// TwinCAT 3 PLC project SDSPLC
// Title: SDS M2
// Company: Aperture Science
// Author: A. Wallace
// ProjectVersion: 0.0.0
// ProgramVersion: 3.1.4022.2
// libraries:
//   Tc2_Standard, * (Beckhoff Automation GmbH)
//   Tc2_System, * (Beckhoff Automation GmbH)
//   Tc3_Module, * (Beckhoff Automation GmbH)
//   LCLS General,0.1.2,SLAC
//   LCLSVacuumLib,1.12.6969,SLAC
//   Tc2_EtherCAT,3.3.13.0,Beckhoff Automation GmbH
//   Tc2_IoFunctions,3.3.11.0,Beckhoff Automation GmbH
//   Tc2_MC2,3.3.37.0,Beckhoff Automation GmbH
//   Tc2_ModbusSrv,3.3.1.0,Beckhoff Automation GmbH
//   Tc2_SerialCom,3.3.6.0,Beckhoff Automation GmbH
//   Tc2_SUPS,3.3.6.0,Beckhoff Automation GmbH
//   Tc2_Utilities,3.3.35.0,Beckhoff Automation GmbH
// project tree:
//   DUTs/ALI/ E_AxisMoveMode.TcDUT (not stored), E_CTRL_MODE.TcDUT (not stored), E_PropValveFBState.TcDUT (not stored), HMI_PropValveCtrlState.TcDUT (not stored), ST_ALI.TcDUT (not stored), ST_ManipAxis.TcDUT (not stored), ST_PIDParams.TcDUT (not stored), ST_PressureController.TcDUT (not stored), ST_PropValveMKS253.TcDUT (not stored)
//   DUTs/Bronkhorst/ E_BHElFlowUnit.TcDUT (not stored), ST_BhElFlow.TcDUT (not stored), ST_BhFMControl.TcDUT (not stored), ST_BhFMStatus.TcDUT (not stored)
//   DUTs/ E_AxisMotionState.TcDUT (not stored), ST_M3GasManifold.TcDUT (not stored), ST_ManifoldValve.TcDUT (not stored), ST_Proportionair.TcDUT (not stored), ST_RegDeadbandControls.TcDUT (not stored), ST_Regulator.TcDUT (not stored), ST_Selector.TcDUT (not stored), ST_SelectorM3.TcDUT (not stored), ST_SensirionFM.TcDUT (not stored), ST_Shaker.TcDUT (not stored), ST_ShakerControls.TcDUT (not stored)
//   DUTs/IO_Structs/ ST_ALIIO.TcDUT (not stored), ST_M2SelectorIO.TcDUT (not stored), ST_M3DeviceBaseIO.TcDUT (not stored), ST_M3GasManifoldIO.TcDUT (not stored), ST_M3PressCtrlIO.TcDUT (not stored), ST_M3SelectorIO.TcDUT (not stored)
//   DUTs/Sensirion/ ST_SensirionFMControl.TcDUT (not stored), ST_SensirionFMStatus.TcDUT (not stored)
//   DUTs/TEC/ ST_TECControl.TcDUT (not stored), ST_TECStatus.TcDUT (not stored)
//   DUTs/Vici/ ST_ViciControl.TcDUT (not stored), ST_ViciStatus.TcDUT (not stored)
//   GVLs/ GVL.TcGVL (not stored), GVL_Autosave.TcGVL (not stored), GVL_ComBuffers.TcGVL (not stored), GVL_Devices.TcGVL (not stored), GVL_IO.TcGVL (not stored), GVL_misc.TcGVL (not stored)
//   / PlcTask.TcTTO (not stored), SerialComm.TcTTO (not stored)
//   POUs/ALI/ FB_ALI.TcPOU (not stored), FB_PID_EXT.TcPOU (not stored), MC_SmoothMover.TcPOU (not stored), F_AxisRef_To_MSTA.TcPOU (not stored), FB_ManipAxis.TcPOU (not stored), FB_PropValve.TcPOU (not stored)
//   POUs/Bronkhorst/ FB_L01Driver.TcPOU (not stored), FB_FlowBusTransaction.TcPOU (not stored)
//   POUs/ FB_SelectorM3.TcPOU (not stored), MAIN.TcPOU (not stored), p_ALI.TcPOU (not stored), p_Autosave.TcPOU (not stored), p_AutoWash.TcPOU (not stored), p_CoolerShaker.TcPOU (not stored), p_ESTOP.TcPOU (not stored), p_Manifold.TcPOU (not stored), p_ModbusRx.TcPOU (not stored), p_ModbusTx.TcPOU (not stored), p_Regulators.TcPOU (not stored), p_SampleSelector.TcPOU (not stored), p_SampleSelector2.TcPOU (not stored), p_Shakers.TcPOU (not stored), p_SoftIO.TcPOU (not stored), p_VacGaugeSup.TcPOU (not stored), SerialTxRx.TcPOU (not stored), p_StatusLights.TcPOU (not stored)
//   POUs/Helpers/ FB_EcatDiag.TcPOU (not stored), FB_ManiValve.TcPOU (not stored), FB_SelectorSync.TcPOU (not stored), FB_ShiftByteArray.TcPOU (not stored)
//   POUs/Regulators/ FB_ProportionairRegulator.TcPOU (not stored), FB_Regulator.TcPOU (not stored), F_rPressure.TcPOU (not stored)
//   POUs/Sensirion/ FB_SensirionDriver.TcPOU (not stored), FB_SensirionTransaction.TcPOU (not stored), fSHDLCChecksum.TcPOU (not stored)
//   POUs/TEC/ FB_TECDriver.TcPOU (not stored), FB_TECTransaction.TcPOU (not stored)
//   POUs/VICI/ FB_ViciDriver.TcPOU, FB_ViciTransaction.TcPOU (not stored)
//   VISUs/ Main.TcVIS (not stored)
// real-time tasks:
//   TASK SerialComm: cycle T#5ms, priority 1, ADS port 350
//   TASK PlcTask: cycle T#10ms, priority 20, ADS port 351
// motion (NC):
// I/O:
//   DEVICE MAIN (EtherCAT)
// variable links:
//   SDSPLC Instance <-> MAIN (EtherCAT)
//     PlcTask Inputs/GVL.g_aEcatMaster1 <-> InfoData/AmsNetId
//     PlcTask Inputs/GVL_IO.iq_stPressCtrlA.i_SyncUnitWC <-> SyncUnits/[PCM A (EP1111)]/<unreferenced>/WcState/WcState
//   SDSPLC Instance <-> MAIN (EtherCAT)/ALI_Gauges (EP3174-0002)
//     PlcTask Inputs/GVL_Devices.stALI.i_EP3174_Ch{1..4} <-> AI Standard Channel {1..4}/Value  (4 links)
//   SDSPLC Instance <-> MAIN (EtherCAT)/ALI_PropValve (EP7041-0002)
//     PlcTask Inputs/GVL_Devices.stALI.stPropVlv.i_HLS <-> STM Status/Status/Digital input 1
//     PlcTask Inputs/GVL_Devices.stALI.stPropVlv.i_LLS <-> STM Status/Status/Digital input 2
//   SDSPLC Instance <-> MAIN (EtherCAT)/ALI_X (EP7041-0002)
//     PlcTask Inputs/GVL_Devices.stALI.axisX.xHiLS <-> STM Status/Status/Digital input 2
//     PlcTask Inputs/GVL_Devices.stALI.axisX.xLoLS <-> STM Status/Status/Digital input 1
//   SDSPLC Instance <-> MAIN (EtherCAT)/ALI_Y (EP7041-0002)
//     PlcTask Inputs/GVL_Devices.stALI.axisY.xHiLS <-> STM Status/Status/Digital input 2
//     PlcTask Inputs/GVL_Devices.stALI.axisY.xLoLS <-> STM Status/Status/Digital input 1
//   SDSPLC Instance <-> MAIN (EtherCAT)/ALI_Z (EP7041-0002)
//     PlcTask Inputs/GVL_Devices.stALI.axisZ.xHiLS <-> STM Status/Status/Digital input 2
//     PlcTask Inputs/GVL_Devices.stALI.axisZ.xLoLS <-> STM Status/Status/Digital input 1
//   SDSPLC Instance <-> MAIN (EtherCAT)/Gas_Mani_NeedleValve (EP4374-0002)
//     PlcTask Inputs/GVL_IO.iq_stM3GasManifold.i_EP4374_Ch1 <-> AI Inputs Channel 1/Value
//     PlcTask Inputs/GVL_IO.iq_stM3GasManifold.i_EP4374_Ch2 <-> AI Inputs Channel 2/Value
//     PlcTask Outputs/GVL_IO.iq_stM3GasManifold.q_EP4374_Ch3 <-> AO Outputs Channel 3/Analog output
//     PlcTask Outputs/GVL_IO.iq_stM3GasManifold.q_EP4374_Ch4 <-> AO Outputs Channel 4/Analog output
//   SDSPLC Instance <-> MAIN (EtherCAT)/Gas_Mani_ValveCtrl (EP2338-0001)
//     PlcTask Outputs/GVL_IO.iq_stM3GasManifold.q_EP2338_Ch{1..8} <-> Channel {9..16}/Output  (8 links)
//   SDSPLC Instance <-> MAIN (EtherCAT)/Gas_Mani_ValveRbk (EP2338-0001)
//     PlcTask Inputs/GVL_IO.iq_stM3GasManifold.i_EP2338_Ch{1..8} <-> Channel {1..8}/Input  (8 links)
//   SDSPLC Instance <-> MAIN (EtherCAT)/M2 Selector A (EP2338-0001)
//     PlcTask Inputs/GVL_IO.iq_stM2SelectorA.i_EP2338_Ch{5..8} <-> Channel {5..8}/Input  (4 links)
//     PlcTask Outputs/GVL_IO.iq_stM2SelectorA.q_EP2338_Ch{1..4} <-> Channel {9..12}/Output  (4 links)
//   SDSPLC Instance <-> MAIN (EtherCAT)/M2 Selector A (EP6002-0002)
//     SerialComm Inputs/GVL_IO.iq_stM2SelectorA.stComIn_EP6002P1/D[0] <-> COM TxPDO-Map Inputs Channel 1/Data In 0
//     SerialComm Inputs/GVL_IO.iq_stM2SelectorA.stComIn_EP6002P1/D[10] <-> COM TxPDO-Map Inputs Channel 1/Data In 10
//     SerialComm Inputs/GVL_IO.iq_stM2SelectorA.stComIn_EP6002P1/D[11] <-> COM TxPDO-Map Inputs Channel 1/Data In 11
//     SerialComm Inputs/GVL_IO.iq_stM2SelectorA.stComIn_EP6002P1/D[12] <-> COM TxPDO-Map Inputs Channel 1/Data In 12
//     SerialComm Inputs/GVL_IO.iq_stM2SelectorA.stComIn_EP6002P1/D[13] <-> COM TxPDO-Map Inputs Channel 1/Data In 13
//     SerialComm Inputs/GVL_IO.iq_stM2SelectorA.stComIn_EP6002P1/D[14] <-> COM TxPDO-Map Inputs Channel 1/Data In 14
//     SerialComm Inputs/GVL_IO.iq_stM2SelectorA.stComIn_EP6002P1/D[15] <-> COM TxPDO-Map Inputs Channel 1/Data In 15
//     SerialComm Inputs/GVL_IO.iq_stM2SelectorA.stComIn_EP6002P1/D[16] <-> COM TxPDO-Map Inputs Channel 1/Data In 16
//     SerialComm Inputs/GVL_IO.iq_stM2SelectorA.stComIn_EP6002P1/D[17] <-> COM TxPDO-Map Inputs Channel 1/Data In 17
//     SerialComm Inputs/GVL_IO.iq_stM2SelectorA.stComIn_EP6002P1/D[18] <-> COM TxPDO-Map Inputs Channel 1/Data In 18
//     SerialComm Inputs/GVL_IO.iq_stM2SelectorA.stComIn_EP6002P1/D[19] <-> COM TxPDO-Map Inputs Channel 1/Data In 19
//     SerialComm Inputs/GVL_IO.iq_stM2SelectorA.stComIn_EP6002P1/D[1] <-> COM TxPDO-Map Inputs Channel 1/Data In 1
//     SerialComm Inputs/GVL_IO.iq_stM2SelectorA.stComIn_EP6002P1/D[20] <-> COM TxPDO-Map Inputs Channel 1/Data In 20
//     SerialComm Inputs/GVL_IO.iq_stM2SelectorA.stComIn_EP6002P1/D[21] <-> COM TxPDO-Map Inputs Channel 1/Data In 21
//     SerialComm Inputs/GVL_IO.iq_stM2SelectorA.stComIn_EP6002P1/D[2] <-> COM TxPDO-Map Inputs Channel 1/Data In 2
//     SerialComm Inputs/GVL_IO.iq_stM2SelectorA.stComIn_EP6002P1/D[3] <-> COM TxPDO-Map Inputs Channel 1/Data In 3
//     SerialComm Inputs/GVL_IO.iq_stM2SelectorA.stComIn_EP6002P1/D[4] <-> COM TxPDO-Map Inputs Channel 1/Data In 4
//     SerialComm Inputs/GVL_IO.iq_stM2SelectorA.stComIn_EP6002P1/D[5] <-> COM TxPDO-Map Inputs Channel 1/Data In 5
//     SerialComm Inputs/GVL_IO.iq_stM2SelectorA.stComIn_EP6002P1/D[6] <-> COM TxPDO-Map Inputs Channel 1/Data In 6
//     SerialComm Inputs/GVL_IO.iq_stM2SelectorA.stComIn_EP6002P1/D[7] <-> COM TxPDO-Map Inputs Channel 1/Data In 7
//     SerialComm Inputs/GVL_IO.iq_stM2SelectorA.stComIn_EP6002P1/D[8] <-> COM TxPDO-Map Inputs Channel 1/Data In 8
//     SerialComm Inputs/GVL_IO.iq_stM2SelectorA.stComIn_EP6002P1/D[9] <-> COM TxPDO-Map Inputs Channel 1/Data In 9
//     SerialComm Inputs/GVL_IO.iq_stM2SelectorA.stComIn_EP6002P2/D[0] <-> COM TxPDO-Map Inputs Channel 2/Data In 0
//     SerialComm Inputs/GVL_IO.iq_stM2SelectorA.stComIn_EP6002P2/D[10] <-> COM TxPDO-Map Inputs Channel 2/Data In 10
//     SerialComm Inputs/GVL_IO.iq_stM2SelectorA.stComIn_EP6002P2/D[11] <-> COM TxPDO-Map Inputs Channel 2/Data In 11
//     SerialComm Inputs/GVL_IO.iq_stM2SelectorA.stComIn_EP6002P2/D[12] <-> COM TxPDO-Map Inputs Channel 2/Data In 12
//     SerialComm Inputs/GVL_IO.iq_stM2SelectorA.stComIn_EP6002P2/D[13] <-> COM TxPDO-Map Inputs Channel 2/Data In 13
//     SerialComm Inputs/GVL_IO.iq_stM2SelectorA.stComIn_EP6002P2/D[14] <-> COM TxPDO-Map Inputs Channel 2/Data In 14
//     SerialComm Inputs/GVL_IO.iq_stM2SelectorA.stComIn_EP6002P2/D[15] <-> COM TxPDO-Map Inputs Channel 2/Data In 15
//     SerialComm Inputs/GVL_IO.iq_stM2SelectorA.stComIn_EP6002P2/D[16] <-> COM TxPDO-Map Inputs Channel 2/Data In 16
//     SerialComm Inputs/GVL_IO.iq_stM2SelectorA.stComIn_EP6002P2/D[17] <-> COM TxPDO-Map Inputs Channel 2/Data In 17
//     SerialComm Inputs/GVL_IO.iq_stM2SelectorA.stComIn_EP6002P2/D[18] <-> COM TxPDO-Map Inputs Channel 2/Data In 18
//     SerialComm Inputs/GVL_IO.iq_stM2SelectorA.stComIn_EP6002P2/D[19] <-> COM TxPDO-Map Inputs Channel 2/Data In 19
//     SerialComm Inputs/GVL_IO.iq_stM2SelectorA.stComIn_EP6002P2/D[1] <-> COM TxPDO-Map Inputs Channel 2/Data In 1
//     SerialComm Inputs/GVL_IO.iq_stM2SelectorA.stComIn_EP6002P2/D[20] <-> COM TxPDO-Map Inputs Channel 2/Data In 20
//     SerialComm Inputs/GVL_IO.iq_stM2SelectorA.stComIn_EP6002P2/D[21] <-> COM TxPDO-Map Inputs Channel 2/Data In 21
//     SerialComm Inputs/GVL_IO.iq_stM2SelectorA.stComIn_EP6002P2/D[2] <-> COM TxPDO-Map Inputs Channel 2/Data In 2
//     SerialComm Inputs/GVL_IO.iq_stM2SelectorA.stComIn_EP6002P2/D[3] <-> COM TxPDO-Map Inputs Channel 2/Data In 3
//     SerialComm Inputs/GVL_IO.iq_stM2SelectorA.stComIn_EP6002P2/D[4] <-> COM TxPDO-Map Inputs Channel 2/Data In 4
//     SerialComm Inputs/GVL_IO.iq_stM2SelectorA.stComIn_EP6002P2/D[5] <-> COM TxPDO-Map Inputs Channel 2/Data In 5
//     SerialComm Inputs/GVL_IO.iq_stM2SelectorA.stComIn_EP6002P2/D[6] <-> COM TxPDO-Map Inputs Channel 2/Data In 6
//     SerialComm Inputs/GVL_IO.iq_stM2SelectorA.stComIn_EP6002P2/D[7] <-> COM TxPDO-Map Inputs Channel 2/Data In 7
//     SerialComm Inputs/GVL_IO.iq_stM2SelectorA.stComIn_EP6002P2/D[8] <-> COM TxPDO-Map Inputs Channel 2/Data In 8
//     SerialComm Inputs/GVL_IO.iq_stM2SelectorA.stComIn_EP6002P2/D[9] <-> COM TxPDO-Map Inputs Channel 2/Data In 9
//     SerialComm Inputs/GVL_IO.iq_stM2SelectorA.stComIn_EP6002P1/Status <-> COM TxPDO-Map Inputs Channel 1/Status
//     SerialComm Inputs/GVL_IO.iq_stM2SelectorA.stComIn_EP6002P2/Status <-> COM TxPDO-Map Inputs Channel 2/Status
//     SerialComm Outputs/GVL_IO.iq_stM2SelectorA.stComOut_EP6002P1/Ctrl <-> COM RxPDO-Map Outputs Channel 1/Ctrl
//     SerialComm Outputs/GVL_IO.iq_stM2SelectorA.stComOut_EP6002P2/Ctrl <-> COM RxPDO-Map Outputs Channel 2/Ctrl
//     SerialComm Outputs/GVL_IO.iq_stM2SelectorA.stComOut_EP6002P1/D[0] <-> COM RxPDO-Map Outputs Channel 1/Data Out 0
//     SerialComm Outputs/GVL_IO.iq_stM2SelectorA.stComOut_EP6002P1/D[10] <-> COM RxPDO-Map Outputs Channel 1/Data Out 10
//     SerialComm Outputs/GVL_IO.iq_stM2SelectorA.stComOut_EP6002P1/D[11] <-> COM RxPDO-Map Outputs Channel 1/Data Out 11
//     SerialComm Outputs/GVL_IO.iq_stM2SelectorA.stComOut_EP6002P1/D[12] <-> COM RxPDO-Map Outputs Channel 1/Data Out 12
//     SerialComm Outputs/GVL_IO.iq_stM2SelectorA.stComOut_EP6002P1/D[13] <-> COM RxPDO-Map Outputs Channel 1/Data Out 13
//     SerialComm Outputs/GVL_IO.iq_stM2SelectorA.stComOut_EP6002P1/D[14] <-> COM RxPDO-Map Outputs Channel 1/Data Out 14
//     SerialComm Outputs/GVL_IO.iq_stM2SelectorA.stComOut_EP6002P1/D[15] <-> COM RxPDO-Map Outputs Channel 1/Data Out 15
//     SerialComm Outputs/GVL_IO.iq_stM2SelectorA.stComOut_EP6002P1/D[16] <-> COM RxPDO-Map Outputs Channel 1/Data Out 16
//     SerialComm Outputs/GVL_IO.iq_stM2SelectorA.stComOut_EP6002P1/D[17] <-> COM RxPDO-Map Outputs Channel 1/Data Out 17
//     SerialComm Outputs/GVL_IO.iq_stM2SelectorA.stComOut_EP6002P1/D[18] <-> COM RxPDO-Map Outputs Channel 1/Data Out 18
//     SerialComm Outputs/GVL_IO.iq_stM2SelectorA.stComOut_EP6002P1/D[19] <-> COM RxPDO-Map Outputs Channel 1/Data Out 19
//     SerialComm Outputs/GVL_IO.iq_stM2SelectorA.stComOut_EP6002P1/D[1] <-> COM RxPDO-Map Outputs Channel 1/Data Out 1
//     SerialComm Outputs/GVL_IO.iq_stM2SelectorA.stComOut_EP6002P1/D[20] <-> COM RxPDO-Map Outputs Channel 1/Data Out 20
//     SerialComm Outputs/GVL_IO.iq_stM2SelectorA.stComOut_EP6002P1/D[21] <-> COM RxPDO-Map Outputs Channel 1/Data Out 21
//     SerialComm Outputs/GVL_IO.iq_stM2SelectorA.stComOut_EP6002P1/D[2] <-> COM RxPDO-Map Outputs Channel 1/Data Out 2
//     SerialComm Outputs/GVL_IO.iq_stM2SelectorA.stComOut_EP6002P1/D[3] <-> COM RxPDO-Map Outputs Channel 1/Data Out 3
//     SerialComm Outputs/GVL_IO.iq_stM2SelectorA.stComOut_EP6002P1/D[4] <-> COM RxPDO-Map Outputs Channel 1/Data Out 4
//     SerialComm Outputs/GVL_IO.iq_stM2SelectorA.stComOut_EP6002P1/D[5] <-> COM RxPDO-Map Outputs Channel 1/Data Out 5
//     SerialComm Outputs/GVL_IO.iq_stM2SelectorA.stComOut_EP6002P1/D[6] <-> COM RxPDO-Map Outputs Channel 1/Data Out 6
//     SerialComm Outputs/GVL_IO.iq_stM2SelectorA.stComOut_EP6002P1/D[7] <-> COM RxPDO-Map Outputs Channel 1/Data Out 7
//     SerialComm Outputs/GVL_IO.iq_stM2SelectorA.stComOut_EP6002P1/D[8] <-> COM RxPDO-Map Outputs Channel 1/Data Out 8
//     SerialComm Outputs/GVL_IO.iq_stM2SelectorA.stComOut_EP6002P1/D[9] <-> COM RxPDO-Map Outputs Channel 1/Data Out 9
//     SerialComm Outputs/GVL_IO.iq_stM2SelectorA.stComOut_EP6002P2/D[0] <-> COM RxPDO-Map Outputs Channel 2/Data Out 0
//     SerialComm Outputs/GVL_IO.iq_stM2SelectorA.stComOut_EP6002P2/D[10] <-> COM RxPDO-Map Outputs Channel 2/Data Out 10
//     SerialComm Outputs/GVL_IO.iq_stM2SelectorA.stComOut_EP6002P2/D[11] <-> COM RxPDO-Map Outputs Channel 2/Data Out 11
//     SerialComm Outputs/GVL_IO.iq_stM2SelectorA.stComOut_EP6002P2/D[12] <-> COM RxPDO-Map Outputs Channel 2/Data Out 12
//     SerialComm Outputs/GVL_IO.iq_stM2SelectorA.stComOut_EP6002P2/D[13] <-> COM RxPDO-Map Outputs Channel 2/Data Out 13
//     SerialComm Outputs/GVL_IO.iq_stM2SelectorA.stComOut_EP6002P2/D[14] <-> COM RxPDO-Map Outputs Channel 2/Data Out 14
//     SerialComm Outputs/GVL_IO.iq_stM2SelectorA.stComOut_EP6002P2/D[15] <-> COM RxPDO-Map Outputs Channel 2/Data Out 15
//     SerialComm Outputs/GVL_IO.iq_stM2SelectorA.stComOut_EP6002P2/D[16] <-> COM RxPDO-Map Outputs Channel 2/Data Out 16
//     SerialComm Outputs/GVL_IO.iq_stM2SelectorA.stComOut_EP6002P2/D[17] <-> COM RxPDO-Map Outputs Channel 2/Data Out 17
//     SerialComm Outputs/GVL_IO.iq_stM2SelectorA.stComOut_EP6002P2/D[18] <-> COM RxPDO-Map Outputs Channel 2/Data Out 18
//     SerialComm Outputs/GVL_IO.iq_stM2SelectorA.stComOut_EP6002P2/D[19] <-> COM RxPDO-Map Outputs Channel 2/Data Out 19
//     SerialComm Outputs/GVL_IO.iq_stM2SelectorA.stComOut_EP6002P2/D[1] <-> COM RxPDO-Map Outputs Channel 2/Data Out 1
//     SerialComm Outputs/GVL_IO.iq_stM2SelectorA.stComOut_EP6002P2/D[20] <-> COM RxPDO-Map Outputs Channel 2/Data Out 20
//     SerialComm Outputs/GVL_IO.iq_stM2SelectorA.stComOut_EP6002P2/D[21] <-> COM RxPDO-Map Outputs Channel 2/Data Out 21
//     SerialComm Outputs/GVL_IO.iq_stM2SelectorA.stComOut_EP6002P2/D[2] <-> COM RxPDO-Map Outputs Channel 2/Data Out 2
//     SerialComm Outputs/GVL_IO.iq_stM2SelectorA.stComOut_EP6002P2/D[3] <-> COM RxPDO-Map Outputs Channel 2/Data Out 3
//     SerialComm Outputs/GVL_IO.iq_stM2SelectorA.stComOut_EP6002P2/D[4] <-> COM RxPDO-Map Outputs Channel 2/Data Out 4
//     SerialComm Outputs/GVL_IO.iq_stM2SelectorA.stComOut_EP6002P2/D[5] <-> COM RxPDO-Map Outputs Channel 2/Data Out 5
//     SerialComm Outputs/GVL_IO.iq_stM2SelectorA.stComOut_EP6002P2/D[6] <-> COM RxPDO-Map Outputs Channel 2/Data Out 6
//     SerialComm Outputs/GVL_IO.iq_stM2SelectorA.stComOut_EP6002P2/D[7] <-> COM RxPDO-Map Outputs Channel 2/Data Out 7
//     SerialComm Outputs/GVL_IO.iq_stM2SelectorA.stComOut_EP6002P2/D[8] <-> COM RxPDO-Map Outputs Channel 2/Data Out 8
//     SerialComm Outputs/GVL_IO.iq_stM2SelectorA.stComOut_EP6002P2/D[9] <-> COM RxPDO-Map Outputs Channel 2/Data Out 9
//   SDSPLC Instance <-> MAIN (EtherCAT)/M2 Selector B (EP2338-0001)
//     PlcTask Inputs/GVL_IO.iq_stM2SelectorB.i_EP2338_Ch{5..8} <-> Channel {5..8}/Input  (4 links)
//     PlcTask Outputs/GVL_IO.iq_stM2SelectorB.q_EP2338_Ch{1..4} <-> Channel {9..12}/Output  (4 links)
//   SDSPLC Instance <-> MAIN (EtherCAT)/M2 Selector B (EP6002-0002)
//     SerialComm Inputs/GVL_IO.iq_stM2SelectorB.stComIn_EP6002P1/D[0] <-> COM TxPDO-Map Inputs Channel 1/Data In 0
//     SerialComm Inputs/GVL_IO.iq_stM2SelectorB.stComIn_EP6002P1/D[10] <-> COM TxPDO-Map Inputs Channel 1/Data In 10
//     SerialComm Inputs/GVL_IO.iq_stM2SelectorB.stComIn_EP6002P1/D[11] <-> COM TxPDO-Map Inputs Channel 1/Data In 11
//     SerialComm Inputs/GVL_IO.iq_stM2SelectorB.stComIn_EP6002P1/D[12] <-> COM TxPDO-Map Inputs Channel 1/Data In 12
//     SerialComm Inputs/GVL_IO.iq_stM2SelectorB.stComIn_EP6002P1/D[13] <-> COM TxPDO-Map Inputs Channel 1/Data In 13
//     SerialComm Inputs/GVL_IO.iq_stM2SelectorB.stComIn_EP6002P1/D[14] <-> COM TxPDO-Map Inputs Channel 1/Data In 14
//     SerialComm Inputs/GVL_IO.iq_stM2SelectorB.stComIn_EP6002P1/D[15] <-> COM TxPDO-Map Inputs Channel 1/Data In 15
//     SerialComm Inputs/GVL_IO.iq_stM2SelectorB.stComIn_EP6002P1/D[16] <-> COM TxPDO-Map Inputs Channel 1/Data In 16
//     SerialComm Inputs/GVL_IO.iq_stM2SelectorB.stComIn_EP6002P1/D[17] <-> COM TxPDO-Map Inputs Channel 1/Data In 17
//     SerialComm Inputs/GVL_IO.iq_stM2SelectorB.stComIn_EP6002P1/D[18] <-> COM TxPDO-Map Inputs Channel 1/Data In 18
//     SerialComm Inputs/GVL_IO.iq_stM2SelectorB.stComIn_EP6002P1/D[19] <-> COM TxPDO-Map Inputs Channel 1/Data In 19
//     SerialComm Inputs/GVL_IO.iq_stM2SelectorB.stComIn_EP6002P1/D[1] <-> COM TxPDO-Map Inputs Channel 1/Data In 1
//     SerialComm Inputs/GVL_IO.iq_stM2SelectorB.stComIn_EP6002P1/D[20] <-> COM TxPDO-Map Inputs Channel 1/Data In 20
//     SerialComm Inputs/GVL_IO.iq_stM2SelectorB.stComIn_EP6002P1/D[21] <-> COM TxPDO-Map Inputs Channel 1/Data In 21
//     SerialComm Inputs/GVL_IO.iq_stM2SelectorB.stComIn_EP6002P1/D[2] <-> COM TxPDO-Map Inputs Channel 1/Data In 2
//     SerialComm Inputs/GVL_IO.iq_stM2SelectorB.stComIn_EP6002P1/D[3] <-> COM TxPDO-Map Inputs Channel 1/Data In 3
//     SerialComm Inputs/GVL_IO.iq_stM2SelectorB.stComIn_EP6002P1/D[4] <-> COM TxPDO-Map Inputs Channel 1/Data In 4
//     SerialComm Inputs/GVL_IO.iq_stM2SelectorB.stComIn_EP6002P1/D[5] <-> COM TxPDO-Map Inputs Channel 1/Data In 5
//     SerialComm Inputs/GVL_IO.iq_stM2SelectorB.stComIn_EP6002P1/D[6] <-> COM TxPDO-Map Inputs Channel 1/Data In 6
//     SerialComm Inputs/GVL_IO.iq_stM2SelectorB.stComIn_EP6002P1/D[7] <-> COM TxPDO-Map Inputs Channel 1/Data In 7
//     SerialComm Inputs/GVL_IO.iq_stM2SelectorB.stComIn_EP6002P1/D[8] <-> COM TxPDO-Map Inputs Channel 1/Data In 8
//     SerialComm Inputs/GVL_IO.iq_stM2SelectorB.stComIn_EP6002P1/D[9] <-> COM TxPDO-Map Inputs Channel 1/Data In 9
//     SerialComm Inputs/GVL_IO.iq_stM2SelectorB.stComIn_EP6002P2/D[0] <-> COM TxPDO-Map Inputs Channel 2/Data In 0
//     SerialComm Inputs/GVL_IO.iq_stM2SelectorB.stComIn_EP6002P2/D[10] <-> COM TxPDO-Map Inputs Channel 2/Data In 10
//     SerialComm Inputs/GVL_IO.iq_stM2SelectorB.stComIn_EP6002P2/D[11] <-> COM TxPDO-Map Inputs Channel 2/Data In 11
//     SerialComm Inputs/GVL_IO.iq_stM2SelectorB.stComIn_EP6002P2/D[12] <-> COM TxPDO-Map Inputs Channel 2/Data In 12
//     SerialComm Inputs/GVL_IO.iq_stM2SelectorB.stComIn_EP6002P2/D[13] <-> COM TxPDO-Map Inputs Channel 2/Data In 13
//     SerialComm Inputs/GVL_IO.iq_stM2SelectorB.stComIn_EP6002P2/D[14] <-> COM TxPDO-Map Inputs Channel 2/Data In 14
//     SerialComm Inputs/GVL_IO.iq_stM2SelectorB.stComIn_EP6002P2/D[15] <-> COM TxPDO-Map Inputs Channel 2/Data In 15
//     SerialComm Inputs/GVL_IO.iq_stM2SelectorB.stComIn_EP6002P2/D[16] <-> COM TxPDO-Map Inputs Channel 2/Data In 16
//     SerialComm Inputs/GVL_IO.iq_stM2SelectorB.stComIn_EP6002P2/D[17] <-> COM TxPDO-Map Inputs Channel 2/Data In 17
//     SerialComm Inputs/GVL_IO.iq_stM2SelectorB.stComIn_EP6002P2/D[18] <-> COM TxPDO-Map Inputs Channel 2/Data In 18
//     SerialComm Inputs/GVL_IO.iq_stM2SelectorB.stComIn_EP6002P2/D[19] <-> COM TxPDO-Map Inputs Channel 2/Data In 19
//     SerialComm Inputs/GVL_IO.iq_stM2SelectorB.stComIn_EP6002P2/D[1] <-> COM TxPDO-Map Inputs Channel 2/Data In 1
//     SerialComm Inputs/GVL_IO.iq_stM2SelectorB.stComIn_EP6002P2/D[20] <-> COM TxPDO-Map Inputs Channel 2/Data In 20
//     SerialComm Inputs/GVL_IO.iq_stM2SelectorB.stComIn_EP6002P2/D[21] <-> COM TxPDO-Map Inputs Channel 2/Data In 21
//     SerialComm Inputs/GVL_IO.iq_stM2SelectorB.stComIn_EP6002P2/D[2] <-> COM TxPDO-Map Inputs Channel 2/Data In 2
//     SerialComm Inputs/GVL_IO.iq_stM2SelectorB.stComIn_EP6002P2/D[3] <-> COM TxPDO-Map Inputs Channel 2/Data In 3
//     SerialComm Inputs/GVL_IO.iq_stM2SelectorB.stComIn_EP6002P2/D[4] <-> COM TxPDO-Map Inputs Channel 2/Data In 4
//     SerialComm Inputs/GVL_IO.iq_stM2SelectorB.stComIn_EP6002P2/D[5] <-> COM TxPDO-Map Inputs Channel 2/Data In 5
//     SerialComm Inputs/GVL_IO.iq_stM2SelectorB.stComIn_EP6002P2/D[6] <-> COM TxPDO-Map Inputs Channel 2/Data In 6
//     SerialComm Inputs/GVL_IO.iq_stM2SelectorB.stComIn_EP6002P2/D[7] <-> COM TxPDO-Map Inputs Channel 2/Data In 7
//     SerialComm Inputs/GVL_IO.iq_stM2SelectorB.stComIn_EP6002P2/D[8] <-> COM TxPDO-Map Inputs Channel 2/Data In 8
//     SerialComm Inputs/GVL_IO.iq_stM2SelectorB.stComIn_EP6002P2/D[9] <-> COM TxPDO-Map Inputs Channel 2/Data In 9
//     SerialComm Inputs/GVL_IO.iq_stM2SelectorB.stComIn_EP6002P1/Status <-> COM TxPDO-Map Inputs Channel 1/Status
//     SerialComm Inputs/GVL_IO.iq_stM2SelectorB.stComIn_EP6002P2/Status <-> COM TxPDO-Map Inputs Channel 2/Status
//     SerialComm Outputs/GVL_IO.iq_stM2SelectorB.stComOut_EP6002P1/Ctrl <-> COM RxPDO-Map Outputs Channel 1/Ctrl
//     SerialComm Outputs/GVL_IO.iq_stM2SelectorB.stComOut_EP6002P2/Ctrl <-> COM RxPDO-Map Outputs Channel 2/Ctrl
//     SerialComm Outputs/GVL_IO.iq_stM2SelectorB.stComOut_EP6002P1/D[0] <-> COM RxPDO-Map Outputs Channel 1/Data Out 0
//     SerialComm Outputs/GVL_IO.iq_stM2SelectorB.stComOut_EP6002P1/D[10] <-> COM RxPDO-Map Outputs Channel 1/Data Out 10
//     SerialComm Outputs/GVL_IO.iq_stM2SelectorB.stComOut_EP6002P1/D[11] <-> COM RxPDO-Map Outputs Channel 1/Data Out 11
//     SerialComm Outputs/GVL_IO.iq_stM2SelectorB.stComOut_EP6002P1/D[12] <-> COM RxPDO-Map Outputs Channel 1/Data Out 12
//     SerialComm Outputs/GVL_IO.iq_stM2SelectorB.stComOut_EP6002P1/D[13] <-> COM RxPDO-Map Outputs Channel 1/Data Out 13
//     SerialComm Outputs/GVL_IO.iq_stM2SelectorB.stComOut_EP6002P1/D[14] <-> COM RxPDO-Map Outputs Channel 1/Data Out 14
//     SerialComm Outputs/GVL_IO.iq_stM2SelectorB.stComOut_EP6002P1/D[15] <-> COM RxPDO-Map Outputs Channel 1/Data Out 15
//     SerialComm Outputs/GVL_IO.iq_stM2SelectorB.stComOut_EP6002P1/D[16] <-> COM RxPDO-Map Outputs Channel 1/Data Out 16
//     SerialComm Outputs/GVL_IO.iq_stM2SelectorB.stComOut_EP6002P1/D[17] <-> COM RxPDO-Map Outputs Channel 1/Data Out 17
//     SerialComm Outputs/GVL_IO.iq_stM2SelectorB.stComOut_EP6002P1/D[18] <-> COM RxPDO-Map Outputs Channel 1/Data Out 18
//     SerialComm Outputs/GVL_IO.iq_stM2SelectorB.stComOut_EP6002P1/D[19] <-> COM RxPDO-Map Outputs Channel 1/Data Out 19
//     SerialComm Outputs/GVL_IO.iq_stM2SelectorB.stComOut_EP6002P1/D[1] <-> COM RxPDO-Map Outputs Channel 1/Data Out 1
//     SerialComm Outputs/GVL_IO.iq_stM2SelectorB.stComOut_EP6002P1/D[20] <-> COM RxPDO-Map Outputs Channel 1/Data Out 20
//     SerialComm Outputs/GVL_IO.iq_stM2SelectorB.stComOut_EP6002P1/D[21] <-> COM RxPDO-Map Outputs Channel 1/Data Out 21
//     SerialComm Outputs/GVL_IO.iq_stM2SelectorB.stComOut_EP6002P1/D[2] <-> COM RxPDO-Map Outputs Channel 1/Data Out 2
//     SerialComm Outputs/GVL_IO.iq_stM2SelectorB.stComOut_EP6002P1/D[3] <-> COM RxPDO-Map Outputs Channel 1/Data Out 3
//     SerialComm Outputs/GVL_IO.iq_stM2SelectorB.stComOut_EP6002P1/D[4] <-> COM RxPDO-Map Outputs Channel 1/Data Out 4
//     SerialComm Outputs/GVL_IO.iq_stM2SelectorB.stComOut_EP6002P1/D[5] <-> COM RxPDO-Map Outputs Channel 1/Data Out 5
//     SerialComm Outputs/GVL_IO.iq_stM2SelectorB.stComOut_EP6002P1/D[6] <-> COM RxPDO-Map Outputs Channel 1/Data Out 6
//     SerialComm Outputs/GVL_IO.iq_stM2SelectorB.stComOut_EP6002P1/D[7] <-> COM RxPDO-Map Outputs Channel 1/Data Out 7
//     SerialComm Outputs/GVL_IO.iq_stM2SelectorB.stComOut_EP6002P1/D[8] <-> COM RxPDO-Map Outputs Channel 1/Data Out 8
//     SerialComm Outputs/GVL_IO.iq_stM2SelectorB.stComOut_EP6002P1/D[9] <-> COM RxPDO-Map Outputs Channel 1/Data Out 9
//     SerialComm Outputs/GVL_IO.iq_stM2SelectorB.stComOut_EP6002P2/D[0] <-> COM RxPDO-Map Outputs Channel 2/Data Out 0
//     SerialComm Outputs/GVL_IO.iq_stM2SelectorB.stComOut_EP6002P2/D[10] <-> COM RxPDO-Map Outputs Channel 2/Data Out 10
//     SerialComm Outputs/GVL_IO.iq_stM2SelectorB.stComOut_EP6002P2/D[11] <-> COM RxPDO-Map Outputs Channel 2/Data Out 11
//     SerialComm Outputs/GVL_IO.iq_stM2SelectorB.stComOut_EP6002P2/D[12] <-> COM RxPDO-Map Outputs Channel 2/Data Out 12
//     SerialComm Outputs/GVL_IO.iq_stM2SelectorB.stComOut_EP6002P2/D[13] <-> COM RxPDO-Map Outputs Channel 2/Data Out 13
//     SerialComm Outputs/GVL_IO.iq_stM2SelectorB.stComOut_EP6002P2/D[14] <-> COM RxPDO-Map Outputs Channel 2/Data Out 14
//     SerialComm Outputs/GVL_IO.iq_stM2SelectorB.stComOut_EP6002P2/D[15] <-> COM RxPDO-Map Outputs Channel 2/Data Out 15
//     SerialComm Outputs/GVL_IO.iq_stM2SelectorB.stComOut_EP6002P2/D[16] <-> COM RxPDO-Map Outputs Channel 2/Data Out 16
//     SerialComm Outputs/GVL_IO.iq_stM2SelectorB.stComOut_EP6002P2/D[17] <-> COM RxPDO-Map Outputs Channel 2/Data Out 17
//     SerialComm Outputs/GVL_IO.iq_stM2SelectorB.stComOut_EP6002P2/D[18] <-> COM RxPDO-Map Outputs Channel 2/Data Out 18
//     SerialComm Outputs/GVL_IO.iq_stM2SelectorB.stComOut_EP6002P2/D[19] <-> COM RxPDO-Map Outputs Channel 2/Data Out 19
//     SerialComm Outputs/GVL_IO.iq_stM2SelectorB.stComOut_EP6002P2/D[1] <-> COM RxPDO-Map Outputs Channel 2/Data Out 1
//     SerialComm Outputs/GVL_IO.iq_stM2SelectorB.stComOut_EP6002P2/D[20] <-> COM RxPDO-Map Outputs Channel 2/Data Out 20
//     SerialComm Outputs/GVL_IO.iq_stM2SelectorB.stComOut_EP6002P2/D[21] <-> COM RxPDO-Map Outputs Channel 2/Data Out 21
//     SerialComm Outputs/GVL_IO.iq_stM2SelectorB.stComOut_EP6002P2/D[2] <-> COM RxPDO-Map Outputs Channel 2/Data Out 2
//     SerialComm Outputs/GVL_IO.iq_stM2SelectorB.stComOut_EP6002P2/D[3] <-> COM RxPDO-Map Outputs Channel 2/Data Out 3
//     SerialComm Outputs/GVL_IO.iq_stM2SelectorB.stComOut_EP6002P2/D[4] <-> COM RxPDO-Map Outputs Channel 2/Data Out 4
//     SerialComm Outputs/GVL_IO.iq_stM2SelectorB.stComOut_EP6002P2/D[5] <-> COM RxPDO-Map Outputs Channel 2/Data Out 5
//     SerialComm Outputs/GVL_IO.iq_stM2SelectorB.stComOut_EP6002P2/D[6] <-> COM RxPDO-Map Outputs Channel 2/Data Out 6
//     SerialComm Outputs/GVL_IO.iq_stM2SelectorB.stComOut_EP6002P2/D[7] <-> COM RxPDO-Map Outputs Channel 2/Data Out 7
//     SerialComm Outputs/GVL_IO.iq_stM2SelectorB.stComOut_EP6002P2/D[8] <-> COM RxPDO-Map Outputs Channel 2/Data Out 8
//     SerialComm Outputs/GVL_IO.iq_stM2SelectorB.stComOut_EP6002P2/D[9] <-> COM RxPDO-Map Outputs Channel 2/Data Out 9
//   SDSPLC Instance <-> MAIN (EtherCAT)/M3 Selector A Digital IO (EP2338-1001)
//     PlcTask Inputs/GVL_IO.iq_stM3SelectorA.i_EP2338_Ch{5..8} <-> Channel {5..8}/Input  (4 links)
//     PlcTask Outputs/GVL_IO.iq_stM3SelectorA.q_EP2338_Ch{1..4} <-> Channel {9..12}/Output  (4 links)
//   SDSPLC Instance <-> MAIN (EtherCAT)/M3 Selector A Mass Flow Meter (Mass Flow / Pressure Controller - Slave)
//     PlcTask Inputs/GVL_IO.iq_stM3SelectorA.i_RawUnit <-> TxPDO/Unit
//     PlcTask Inputs/GVL_IO.iq_stM3SelectorA.i_mfmFlow <-> TxPDO/fMeasure
//   SDSPLC Instance <-> MAIN (EtherCAT)/M3 Selector A Serial IO (EP6002-0002)
//     PlcTask Inputs/GVL_IO.iq_stM3SelectorA.stComIn_EP6002P1/D[0] <-> COM TxPDO-Map Inputs Channel 1/Data In 0
//     PlcTask Inputs/GVL_IO.iq_stM3SelectorA.stComIn_EP6002P1/D[10] <-> COM TxPDO-Map Inputs Channel 1/Data In 10
//     PlcTask Inputs/GVL_IO.iq_stM3SelectorA.stComIn_EP6002P1/D[11] <-> COM TxPDO-Map Inputs Channel 1/Data In 11
//     PlcTask Inputs/GVL_IO.iq_stM3SelectorA.stComIn_EP6002P1/D[12] <-> COM TxPDO-Map Inputs Channel 1/Data In 12
//     PlcTask Inputs/GVL_IO.iq_stM3SelectorA.stComIn_EP6002P1/D[13] <-> COM TxPDO-Map Inputs Channel 1/Data In 13
//     PlcTask Inputs/GVL_IO.iq_stM3SelectorA.stComIn_EP6002P1/D[14] <-> COM TxPDO-Map Inputs Channel 1/Data In 14
//     PlcTask Inputs/GVL_IO.iq_stM3SelectorA.stComIn_EP6002P1/D[15] <-> COM TxPDO-Map Inputs Channel 1/Data In 15
//     PlcTask Inputs/GVL_IO.iq_stM3SelectorA.stComIn_EP6002P1/D[16] <-> COM TxPDO-Map Inputs Channel 1/Data In 16
//     PlcTask Inputs/GVL_IO.iq_stM3SelectorA.stComIn_EP6002P1/D[17] <-> COM TxPDO-Map Inputs Channel 1/Data In 17
//     PlcTask Inputs/GVL_IO.iq_stM3SelectorA.stComIn_EP6002P1/D[18] <-> COM TxPDO-Map Inputs Channel 1/Data In 18
//     PlcTask Inputs/GVL_IO.iq_stM3SelectorA.stComIn_EP6002P1/D[19] <-> COM TxPDO-Map Inputs Channel 1/Data In 19
//     PlcTask Inputs/GVL_IO.iq_stM3SelectorA.stComIn_EP6002P1/D[1] <-> COM TxPDO-Map Inputs Channel 1/Data In 1
//     PlcTask Inputs/GVL_IO.iq_stM3SelectorA.stComIn_EP6002P1/D[20] <-> COM TxPDO-Map Inputs Channel 1/Data In 20
//     PlcTask Inputs/GVL_IO.iq_stM3SelectorA.stComIn_EP6002P1/D[21] <-> COM TxPDO-Map Inputs Channel 1/Data In 21
//     PlcTask Inputs/GVL_IO.iq_stM3SelectorA.stComIn_EP6002P1/D[2] <-> COM TxPDO-Map Inputs Channel 1/Data In 2
//     PlcTask Inputs/GVL_IO.iq_stM3SelectorA.stComIn_EP6002P1/D[3] <-> COM TxPDO-Map Inputs Channel 1/Data In 3
//     PlcTask Inputs/GVL_IO.iq_stM3SelectorA.stComIn_EP6002P1/D[4] <-> COM TxPDO-Map Inputs Channel 1/Data In 4
//     PlcTask Inputs/GVL_IO.iq_stM3SelectorA.stComIn_EP6002P1/D[5] <-> COM TxPDO-Map Inputs Channel 1/Data In 5
//     PlcTask Inputs/GVL_IO.iq_stM3SelectorA.stComIn_EP6002P1/D[6] <-> COM TxPDO-Map Inputs Channel 1/Data In 6
//     PlcTask Inputs/GVL_IO.iq_stM3SelectorA.stComIn_EP6002P1/D[7] <-> COM TxPDO-Map Inputs Channel 1/Data In 7
//     PlcTask Inputs/GVL_IO.iq_stM3SelectorA.stComIn_EP6002P1/D[8] <-> COM TxPDO-Map Inputs Channel 1/Data In 8
//     PlcTask Inputs/GVL_IO.iq_stM3SelectorA.stComIn_EP6002P1/D[9] <-> COM TxPDO-Map Inputs Channel 1/Data In 9
//     PlcTask Inputs/GVL_IO.iq_stM3SelectorA.stComIn_EP6002P2/D[0] <-> COM TxPDO-Map Inputs Channel 2/Data In 0
//     PlcTask Inputs/GVL_IO.iq_stM3SelectorA.stComIn_EP6002P2/D[10] <-> COM TxPDO-Map Inputs Channel 2/Data In 10
//     PlcTask Inputs/GVL_IO.iq_stM3SelectorA.stComIn_EP6002P2/D[11] <-> COM TxPDO-Map Inputs Channel 2/Data In 11
//     PlcTask Inputs/GVL_IO.iq_stM3SelectorA.stComIn_EP6002P2/D[12] <-> COM TxPDO-Map Inputs Channel 2/Data In 12
//     PlcTask Inputs/GVL_IO.iq_stM3SelectorA.stComIn_EP6002P2/D[13] <-> COM TxPDO-Map Inputs Channel 2/Data In 13
//     PlcTask Inputs/GVL_IO.iq_stM3SelectorA.stComIn_EP6002P2/D[14] <-> COM TxPDO-Map Inputs Channel 2/Data In 14
//     PlcTask Inputs/GVL_IO.iq_stM3SelectorA.stComIn_EP6002P2/D[15] <-> COM TxPDO-Map Inputs Channel 2/Data In 15
//     PlcTask Inputs/GVL_IO.iq_stM3SelectorA.stComIn_EP6002P2/D[16] <-> COM TxPDO-Map Inputs Channel 2/Data In 16
//     PlcTask Inputs/GVL_IO.iq_stM3SelectorA.stComIn_EP6002P2/D[17] <-> COM TxPDO-Map Inputs Channel 2/Data In 17
//     PlcTask Inputs/GVL_IO.iq_stM3SelectorA.stComIn_EP6002P2/D[18] <-> COM TxPDO-Map Inputs Channel 2/Data In 18
//     PlcTask Inputs/GVL_IO.iq_stM3SelectorA.stComIn_EP6002P2/D[19] <-> COM TxPDO-Map Inputs Channel 2/Data In 19
//     PlcTask Inputs/GVL_IO.iq_stM3SelectorA.stComIn_EP6002P2/D[1] <-> COM TxPDO-Map Inputs Channel 2/Data In 1
//     PlcTask Inputs/GVL_IO.iq_stM3SelectorA.stComIn_EP6002P2/D[20] <-> COM TxPDO-Map Inputs Channel 2/Data In 20
//     PlcTask Inputs/GVL_IO.iq_stM3SelectorA.stComIn_EP6002P2/D[21] <-> COM TxPDO-Map Inputs Channel 2/Data In 21
//     PlcTask Inputs/GVL_IO.iq_stM3SelectorA.stComIn_EP6002P2/D[2] <-> COM TxPDO-Map Inputs Channel 2/Data In 2
//     PlcTask Inputs/GVL_IO.iq_stM3SelectorA.stComIn_EP6002P2/D[3] <-> COM TxPDO-Map Inputs Channel 2/Data In 3
//     PlcTask Inputs/GVL_IO.iq_stM3SelectorA.stComIn_EP6002P2/D[4] <-> COM TxPDO-Map Inputs Channel 2/Data In 4
//     PlcTask Inputs/GVL_IO.iq_stM3SelectorA.stComIn_EP6002P2/D[5] <-> COM TxPDO-Map Inputs Channel 2/Data In 5
//     PlcTask Inputs/GVL_IO.iq_stM3SelectorA.stComIn_EP6002P2/D[6] <-> COM TxPDO-Map Inputs Channel 2/Data In 6
//     PlcTask Inputs/GVL_IO.iq_stM3SelectorA.stComIn_EP6002P2/D[7] <-> COM TxPDO-Map Inputs Channel 2/Data In 7
//     PlcTask Inputs/GVL_IO.iq_stM3SelectorA.stComIn_EP6002P2/D[8] <-> COM TxPDO-Map Inputs Channel 2/Data In 8
//     PlcTask Inputs/GVL_IO.iq_stM3SelectorA.stComIn_EP6002P2/D[9] <-> COM TxPDO-Map Inputs Channel 2/Data In 9
//     PlcTask Inputs/GVL_IO.iq_stM3SelectorA.stComIn_EP6002P1/Status <-> COM TxPDO-Map Inputs Channel 1/Status
//     PlcTask Inputs/GVL_IO.iq_stM3SelectorA.stComIn_EP6002P2/Status <-> COM TxPDO-Map Inputs Channel 2/Status
//     PlcTask Outputs/GVL_IO.iq_stM3SelectorA.stComOut_EP6002P1/Ctrl <-> COM RxPDO-Map Outputs Channel 1/Ctrl
//     PlcTask Outputs/GVL_IO.iq_stM3SelectorA.stComOut_EP6002P2/Ctrl <-> COM RxPDO-Map Outputs Channel 2/Ctrl
//     PlcTask Outputs/GVL_IO.iq_stM3SelectorA.stComOut_EP6002P1/D[0] <-> COM RxPDO-Map Outputs Channel 1/Data Out 0
//     PlcTask Outputs/GVL_IO.iq_stM3SelectorA.stComOut_EP6002P1/D[10] <-> COM RxPDO-Map Outputs Channel 1/Data Out 10
//     PlcTask Outputs/GVL_IO.iq_stM3SelectorA.stComOut_EP6002P1/D[11] <-> COM RxPDO-Map Outputs Channel 1/Data Out 11
//     PlcTask Outputs/GVL_IO.iq_stM3SelectorA.stComOut_EP6002P1/D[12] <-> COM RxPDO-Map Outputs Channel 1/Data Out 12
//     PlcTask Outputs/GVL_IO.iq_stM3SelectorA.stComOut_EP6002P1/D[13] <-> COM RxPDO-Map Outputs Channel 1/Data Out 13
//     PlcTask Outputs/GVL_IO.iq_stM3SelectorA.stComOut_EP6002P1/D[14] <-> COM RxPDO-Map Outputs Channel 1/Data Out 14
//     PlcTask Outputs/GVL_IO.iq_stM3SelectorA.stComOut_EP6002P1/D[15] <-> COM RxPDO-Map Outputs Channel 1/Data Out 15
//     PlcTask Outputs/GVL_IO.iq_stM3SelectorA.stComOut_EP6002P1/D[16] <-> COM RxPDO-Map Outputs Channel 1/Data Out 16
//     PlcTask Outputs/GVL_IO.iq_stM3SelectorA.stComOut_EP6002P1/D[17] <-> COM RxPDO-Map Outputs Channel 1/Data Out 17
//     PlcTask Outputs/GVL_IO.iq_stM3SelectorA.stComOut_EP6002P1/D[18] <-> COM RxPDO-Map Outputs Channel 1/Data Out 18
//     PlcTask Outputs/GVL_IO.iq_stM3SelectorA.stComOut_EP6002P1/D[19] <-> COM RxPDO-Map Outputs Channel 1/Data Out 19
//     PlcTask Outputs/GVL_IO.iq_stM3SelectorA.stComOut_EP6002P1/D[1] <-> COM RxPDO-Map Outputs Channel 1/Data Out 1
//     PlcTask Outputs/GVL_IO.iq_stM3SelectorA.stComOut_EP6002P1/D[20] <-> COM RxPDO-Map Outputs Channel 1/Data Out 20
//     PlcTask Outputs/GVL_IO.iq_stM3SelectorA.stComOut_EP6002P1/D[21] <-> COM RxPDO-Map Outputs Channel 1/Data Out 21
//     PlcTask Outputs/GVL_IO.iq_stM3SelectorA.stComOut_EP6002P1/D[2] <-> COM RxPDO-Map Outputs Channel 1/Data Out 2
//     PlcTask Outputs/GVL_IO.iq_stM3SelectorA.stComOut_EP6002P1/D[3] <-> COM RxPDO-Map Outputs Channel 1/Data Out 3
//     PlcTask Outputs/GVL_IO.iq_stM3SelectorA.stComOut_EP6002P1/D[4] <-> COM RxPDO-Map Outputs Channel 1/Data Out 4
//     PlcTask Outputs/GVL_IO.iq_stM3SelectorA.stComOut_EP6002P1/D[5] <-> COM RxPDO-Map Outputs Channel 1/Data Out 5
//     PlcTask Outputs/GVL_IO.iq_stM3SelectorA.stComOut_EP6002P1/D[6] <-> COM RxPDO-Map Outputs Channel 1/Data Out 6
//     PlcTask Outputs/GVL_IO.iq_stM3SelectorA.stComOut_EP6002P1/D[7] <-> COM RxPDO-Map Outputs Channel 1/Data Out 7
//     PlcTask Outputs/GVL_IO.iq_stM3SelectorA.stComOut_EP6002P1/D[8] <-> COM RxPDO-Map Outputs Channel 1/Data Out 8
//     PlcTask Outputs/GVL_IO.iq_stM3SelectorA.stComOut_EP6002P1/D[9] <-> COM RxPDO-Map Outputs Channel 1/Data Out 9
//     PlcTask Outputs/GVL_IO.iq_stM3SelectorA.stComOut_EP6002P2/D[0] <-> COM RxPDO-Map Outputs Channel 2/Data Out 0
//     PlcTask Outputs/GVL_IO.iq_stM3SelectorA.stComOut_EP6002P2/D[10] <-> COM RxPDO-Map Outputs Channel 2/Data Out 10
//     PlcTask Outputs/GVL_IO.iq_stM3SelectorA.stComOut_EP6002P2/D[11] <-> COM RxPDO-Map Outputs Channel 2/Data Out 11
//     PlcTask Outputs/GVL_IO.iq_stM3SelectorA.stComOut_EP6002P2/D[12] <-> COM RxPDO-Map Outputs Channel 2/Data Out 12
//     PlcTask Outputs/GVL_IO.iq_stM3SelectorA.stComOut_EP6002P2/D[13] <-> COM RxPDO-Map Outputs Channel 2/Data Out 13
//     PlcTask Outputs/GVL_IO.iq_stM3SelectorA.stComOut_EP6002P2/D[14] <-> COM RxPDO-Map Outputs Channel 2/Data Out 14
//     PlcTask Outputs/GVL_IO.iq_stM3SelectorA.stComOut_EP6002P2/D[15] <-> COM RxPDO-Map Outputs Channel 2/Data Out 15
//     PlcTask Outputs/GVL_IO.iq_stM3SelectorA.stComOut_EP6002P2/D[16] <-> COM RxPDO-Map Outputs Channel 2/Data Out 16
//     PlcTask Outputs/GVL_IO.iq_stM3SelectorA.stComOut_EP6002P2/D[17] <-> COM RxPDO-Map Outputs Channel 2/Data Out 17
//     PlcTask Outputs/GVL_IO.iq_stM3SelectorA.stComOut_EP6002P2/D[18] <-> COM RxPDO-Map Outputs Channel 2/Data Out 18
//     PlcTask Outputs/GVL_IO.iq_stM3SelectorA.stComOut_EP6002P2/D[19] <-> COM RxPDO-Map Outputs Channel 2/Data Out 19
//     PlcTask Outputs/GVL_IO.iq_stM3SelectorA.stComOut_EP6002P2/D[1] <-> COM RxPDO-Map Outputs Channel 2/Data Out 1
//     PlcTask Outputs/GVL_IO.iq_stM3SelectorA.stComOut_EP6002P2/D[20] <-> COM RxPDO-Map Outputs Channel 2/Data Out 20
//     PlcTask Outputs/GVL_IO.iq_stM3SelectorA.stComOut_EP6002P2/D[21] <-> COM RxPDO-Map Outputs Channel 2/Data Out 21
//     PlcTask Outputs/GVL_IO.iq_stM3SelectorA.stComOut_EP6002P2/D[2] <-> COM RxPDO-Map Outputs Channel 2/Data Out 2
//     PlcTask Outputs/GVL_IO.iq_stM3SelectorA.stComOut_EP6002P2/D[3] <-> COM RxPDO-Map Outputs Channel 2/Data Out 3
//     PlcTask Outputs/GVL_IO.iq_stM3SelectorA.stComOut_EP6002P2/D[4] <-> COM RxPDO-Map Outputs Channel 2/Data Out 4
//     PlcTask Outputs/GVL_IO.iq_stM3SelectorA.stComOut_EP6002P2/D[5] <-> COM RxPDO-Map Outputs Channel 2/Data Out 5
//     PlcTask Outputs/GVL_IO.iq_stM3SelectorA.stComOut_EP6002P2/D[6] <-> COM RxPDO-Map Outputs Channel 2/Data Out 6
//     PlcTask Outputs/GVL_IO.iq_stM3SelectorA.stComOut_EP6002P2/D[7] <-> COM RxPDO-Map Outputs Channel 2/Data Out 7
//     PlcTask Outputs/GVL_IO.iq_stM3SelectorA.stComOut_EP6002P2/D[8] <-> COM RxPDO-Map Outputs Channel 2/Data Out 8
//     PlcTask Outputs/GVL_IO.iq_stM3SelectorA.stComOut_EP6002P2/D[9] <-> COM RxPDO-Map Outputs Channel 2/Data Out 9
//   SDSPLC Instance <-> MAIN (EtherCAT)/M3 Selector B Digital IO (EP2338-1001)
//     PlcTask Inputs/GVL_IO.iq_stM3SelectorB.i_EP2338_Ch{5..8} <-> Channel {5..8}/Input  (4 links)
//     PlcTask Outputs/GVL_IO.iq_stM3SelectorB.q_EP2338_Ch{1..4} <-> Channel {9..12}/Output  (4 links)
//   SDSPLC Instance <-> MAIN (EtherCAT)/M3 Selector B Mass Flow Meter (Mass Flow / Pressure Controller - Slave)
//     PlcTask Inputs/GVL_IO.iq_stM3SelectorB.i_RawUnit <-> TxPDO/Unit
//     PlcTask Inputs/GVL_IO.iq_stM3SelectorB.i_mfmFlow <-> TxPDO/fMeasure
//   SDSPLC Instance <-> MAIN (EtherCAT)/M3 Selector B Serial IO (EP6002-0002)
//     PlcTask Inputs/GVL_IO.iq_stM3SelectorB.stComIn_EP6002P1/D[0] <-> COM TxPDO-Map Inputs Channel 1/Data In 0
//     PlcTask Inputs/GVL_IO.iq_stM3SelectorB.stComIn_EP6002P1/D[10] <-> COM TxPDO-Map Inputs Channel 1/Data In 10
//     PlcTask Inputs/GVL_IO.iq_stM3SelectorB.stComIn_EP6002P1/D[11] <-> COM TxPDO-Map Inputs Channel 1/Data In 11
//     PlcTask Inputs/GVL_IO.iq_stM3SelectorB.stComIn_EP6002P1/D[12] <-> COM TxPDO-Map Inputs Channel 1/Data In 12
//     PlcTask Inputs/GVL_IO.iq_stM3SelectorB.stComIn_EP6002P1/D[13] <-> COM TxPDO-Map Inputs Channel 1/Data In 13
//     PlcTask Inputs/GVL_IO.iq_stM3SelectorB.stComIn_EP6002P1/D[14] <-> COM TxPDO-Map Inputs Channel 1/Data In 14
//     PlcTask Inputs/GVL_IO.iq_stM3SelectorB.stComIn_EP6002P1/D[15] <-> COM TxPDO-Map Inputs Channel 1/Data In 15
//     PlcTask Inputs/GVL_IO.iq_stM3SelectorB.stComIn_EP6002P1/D[16] <-> COM TxPDO-Map Inputs Channel 1/Data In 16
//     PlcTask Inputs/GVL_IO.iq_stM3SelectorB.stComIn_EP6002P1/D[17] <-> COM TxPDO-Map Inputs Channel 1/Data In 17
//     PlcTask Inputs/GVL_IO.iq_stM3SelectorB.stComIn_EP6002P1/D[18] <-> COM TxPDO-Map Inputs Channel 1/Data In 18
//     PlcTask Inputs/GVL_IO.iq_stM3SelectorB.stComIn_EP6002P1/D[19] <-> COM TxPDO-Map Inputs Channel 1/Data In 19
//     PlcTask Inputs/GVL_IO.iq_stM3SelectorB.stComIn_EP6002P1/D[1] <-> COM TxPDO-Map Inputs Channel 1/Data In 1
//     PlcTask Inputs/GVL_IO.iq_stM3SelectorB.stComIn_EP6002P1/D[20] <-> COM TxPDO-Map Inputs Channel 1/Data In 20
//     PlcTask Inputs/GVL_IO.iq_stM3SelectorB.stComIn_EP6002P1/D[21] <-> COM TxPDO-Map Inputs Channel 1/Data In 21
//     PlcTask Inputs/GVL_IO.iq_stM3SelectorB.stComIn_EP6002P1/D[2] <-> COM TxPDO-Map Inputs Channel 1/Data In 2
//     PlcTask Inputs/GVL_IO.iq_stM3SelectorB.stComIn_EP6002P1/D[3] <-> COM TxPDO-Map Inputs Channel 1/Data In 3
//     PlcTask Inputs/GVL_IO.iq_stM3SelectorB.stComIn_EP6002P1/D[4] <-> COM TxPDO-Map Inputs Channel 1/Data In 4
//     PlcTask Inputs/GVL_IO.iq_stM3SelectorB.stComIn_EP6002P1/D[5] <-> COM TxPDO-Map Inputs Channel 1/Data In 5
//     PlcTask Inputs/GVL_IO.iq_stM3SelectorB.stComIn_EP6002P1/D[6] <-> COM TxPDO-Map Inputs Channel 1/Data In 6
//     PlcTask Inputs/GVL_IO.iq_stM3SelectorB.stComIn_EP6002P1/D[7] <-> COM TxPDO-Map Inputs Channel 1/Data In 7
//     PlcTask Inputs/GVL_IO.iq_stM3SelectorB.stComIn_EP6002P1/D[8] <-> COM TxPDO-Map Inputs Channel 1/Data In 8
//     PlcTask Inputs/GVL_IO.iq_stM3SelectorB.stComIn_EP6002P1/D[9] <-> COM TxPDO-Map Inputs Channel 1/Data In 9
//     PlcTask Inputs/GVL_IO.iq_stM3SelectorB.stComIn_EP6002P2/D[0] <-> COM TxPDO-Map Inputs Channel 2/Data In 0
//     PlcTask Inputs/GVL_IO.iq_stM3SelectorB.stComIn_EP6002P2/D[10] <-> COM TxPDO-Map Inputs Channel 2/Data In 10
//     PlcTask Inputs/GVL_IO.iq_stM3SelectorB.stComIn_EP6002P2/D[11] <-> COM TxPDO-Map Inputs Channel 2/Data In 11
//     PlcTask Inputs/GVL_IO.iq_stM3SelectorB.stComIn_EP6002P2/D[12] <-> COM TxPDO-Map Inputs Channel 2/Data In 12
//     PlcTask Inputs/GVL_IO.iq_stM3SelectorB.stComIn_EP6002P2/D[13] <-> COM TxPDO-Map Inputs Channel 2/Data In 13
//     PlcTask Inputs/GVL_IO.iq_stM3SelectorB.stComIn_EP6002P2/D[14] <-> COM TxPDO-Map Inputs Channel 2/Data In 14
//     PlcTask Inputs/GVL_IO.iq_stM3SelectorB.stComIn_EP6002P2/D[15] <-> COM TxPDO-Map Inputs Channel 2/Data In 15
//     PlcTask Inputs/GVL_IO.iq_stM3SelectorB.stComIn_EP6002P2/D[16] <-> COM TxPDO-Map Inputs Channel 2/Data In 16
//     PlcTask Inputs/GVL_IO.iq_stM3SelectorB.stComIn_EP6002P2/D[17] <-> COM TxPDO-Map Inputs Channel 2/Data In 17
//     PlcTask Inputs/GVL_IO.iq_stM3SelectorB.stComIn_EP6002P2/D[18] <-> COM TxPDO-Map Inputs Channel 2/Data In 18
//     PlcTask Inputs/GVL_IO.iq_stM3SelectorB.stComIn_EP6002P2/D[19] <-> COM TxPDO-Map Inputs Channel 2/Data In 19
//     PlcTask Inputs/GVL_IO.iq_stM3SelectorB.stComIn_EP6002P2/D[1] <-> COM TxPDO-Map Inputs Channel 2/Data In 1
//     PlcTask Inputs/GVL_IO.iq_stM3SelectorB.stComIn_EP6002P2/D[20] <-> COM TxPDO-Map Inputs Channel 2/Data In 20
//     PlcTask Inputs/GVL_IO.iq_stM3SelectorB.stComIn_EP6002P2/D[21] <-> COM TxPDO-Map Inputs Channel 2/Data In 21
//     PlcTask Inputs/GVL_IO.iq_stM3SelectorB.stComIn_EP6002P2/D[2] <-> COM TxPDO-Map Inputs Channel 2/Data In 2
//     PlcTask Inputs/GVL_IO.iq_stM3SelectorB.stComIn_EP6002P2/D[3] <-> COM TxPDO-Map Inputs Channel 2/Data In 3
//     PlcTask Inputs/GVL_IO.iq_stM3SelectorB.stComIn_EP6002P2/D[4] <-> COM TxPDO-Map Inputs Channel 2/Data In 4
//     PlcTask Inputs/GVL_IO.iq_stM3SelectorB.stComIn_EP6002P2/D[5] <-> COM TxPDO-Map Inputs Channel 2/Data In 5
//     PlcTask Inputs/GVL_IO.iq_stM3SelectorB.stComIn_EP6002P2/D[6] <-> COM TxPDO-Map Inputs Channel 2/Data In 6
//     PlcTask Inputs/GVL_IO.iq_stM3SelectorB.stComIn_EP6002P2/D[7] <-> COM TxPDO-Map Inputs Channel 2/Data In 7
//     PlcTask Inputs/GVL_IO.iq_stM3SelectorB.stComIn_EP6002P2/D[8] <-> COM TxPDO-Map Inputs Channel 2/Data In 8
//     PlcTask Inputs/GVL_IO.iq_stM3SelectorB.stComIn_EP6002P2/D[9] <-> COM TxPDO-Map Inputs Channel 2/Data In 9
//     PlcTask Inputs/GVL_IO.iq_stM3SelectorB.stComIn_EP6002P1/Status <-> COM TxPDO-Map Inputs Channel 1/Status
//     PlcTask Inputs/GVL_IO.iq_stM3SelectorB.stComIn_EP6002P2/Status <-> COM TxPDO-Map Inputs Channel 2/Status
//     PlcTask Outputs/GVL_IO.iq_stM3SelectorB.stComOut_EP6002P1/Ctrl <-> COM RxPDO-Map Outputs Channel 1/Ctrl
//     PlcTask Outputs/GVL_IO.iq_stM3SelectorB.stComOut_EP6002P2/Ctrl <-> COM RxPDO-Map Outputs Channel 2/Ctrl
//     PlcTask Outputs/GVL_IO.iq_stM3SelectorB.stComOut_EP6002P1/D[0] <-> COM RxPDO-Map Outputs Channel 1/Data Out 0
//     PlcTask Outputs/GVL_IO.iq_stM3SelectorB.stComOut_EP6002P1/D[10] <-> COM RxPDO-Map Outputs Channel 1/Data Out 10
//     PlcTask Outputs/GVL_IO.iq_stM3SelectorB.stComOut_EP6002P1/D[11] <-> COM RxPDO-Map Outputs Channel 1/Data Out 11
//     PlcTask Outputs/GVL_IO.iq_stM3SelectorB.stComOut_EP6002P1/D[12] <-> COM RxPDO-Map Outputs Channel 1/Data Out 12
//     PlcTask Outputs/GVL_IO.iq_stM3SelectorB.stComOut_EP6002P1/D[13] <-> COM RxPDO-Map Outputs Channel 1/Data Out 13
//     PlcTask Outputs/GVL_IO.iq_stM3SelectorB.stComOut_EP6002P1/D[14] <-> COM RxPDO-Map Outputs Channel 1/Data Out 14
//     PlcTask Outputs/GVL_IO.iq_stM3SelectorB.stComOut_EP6002P1/D[15] <-> COM RxPDO-Map Outputs Channel 1/Data Out 15
//     PlcTask Outputs/GVL_IO.iq_stM3SelectorB.stComOut_EP6002P1/D[16] <-> COM RxPDO-Map Outputs Channel 1/Data Out 16
//     PlcTask Outputs/GVL_IO.iq_stM3SelectorB.stComOut_EP6002P1/D[17] <-> COM RxPDO-Map Outputs Channel 1/Data Out 17
//     PlcTask Outputs/GVL_IO.iq_stM3SelectorB.stComOut_EP6002P1/D[18] <-> COM RxPDO-Map Outputs Channel 1/Data Out 18
//     PlcTask Outputs/GVL_IO.iq_stM3SelectorB.stComOut_EP6002P1/D[19] <-> COM RxPDO-Map Outputs Channel 1/Data Out 19
//     PlcTask Outputs/GVL_IO.iq_stM3SelectorB.stComOut_EP6002P1/D[1] <-> COM RxPDO-Map Outputs Channel 1/Data Out 1
//     PlcTask Outputs/GVL_IO.iq_stM3SelectorB.stComOut_EP6002P1/D[20] <-> COM RxPDO-Map Outputs Channel 1/Data Out 20
//     PlcTask Outputs/GVL_IO.iq_stM3SelectorB.stComOut_EP6002P1/D[21] <-> COM RxPDO-Map Outputs Channel 1/Data Out 21
//     PlcTask Outputs/GVL_IO.iq_stM3SelectorB.stComOut_EP6002P1/D[2] <-> COM RxPDO-Map Outputs Channel 1/Data Out 2
//     PlcTask Outputs/GVL_IO.iq_stM3SelectorB.stComOut_EP6002P1/D[3] <-> COM RxPDO-Map Outputs Channel 1/Data Out 3
//     PlcTask Outputs/GVL_IO.iq_stM3SelectorB.stComOut_EP6002P1/D[4] <-> COM RxPDO-Map Outputs Channel 1/Data Out 4
//     PlcTask Outputs/GVL_IO.iq_stM3SelectorB.stComOut_EP6002P1/D[5] <-> COM RxPDO-Map Outputs Channel 1/Data Out 5
//     PlcTask Outputs/GVL_IO.iq_stM3SelectorB.stComOut_EP6002P1/D[6] <-> COM RxPDO-Map Outputs Channel 1/Data Out 6
//     PlcTask Outputs/GVL_IO.iq_stM3SelectorB.stComOut_EP6002P1/D[7] <-> COM RxPDO-Map Outputs Channel 1/Data Out 7
//     PlcTask Outputs/GVL_IO.iq_stM3SelectorB.stComOut_EP6002P1/D[8] <-> COM RxPDO-Map Outputs Channel 1/Data Out 8
//     PlcTask Outputs/GVL_IO.iq_stM3SelectorB.stComOut_EP6002P1/D[9] <-> COM RxPDO-Map Outputs Channel 1/Data Out 9
//     PlcTask Outputs/GVL_IO.iq_stM3SelectorB.stComOut_EP6002P2/D[0] <-> COM RxPDO-Map Outputs Channel 2/Data Out 0
//     PlcTask Outputs/GVL_IO.iq_stM3SelectorB.stComOut_EP6002P2/D[10] <-> COM RxPDO-Map Outputs Channel 2/Data Out 10
//     PlcTask Outputs/GVL_IO.iq_stM3SelectorB.stComOut_EP6002P2/D[11] <-> COM RxPDO-Map Outputs Channel 2/Data Out 11
//     PlcTask Outputs/GVL_IO.iq_stM3SelectorB.stComOut_EP6002P2/D[12] <-> COM RxPDO-Map Outputs Channel 2/Data Out 12
//     PlcTask Outputs/GVL_IO.iq_stM3SelectorB.stComOut_EP6002P2/D[13] <-> COM RxPDO-Map Outputs Channel 2/Data Out 13
//     PlcTask Outputs/GVL_IO.iq_stM3SelectorB.stComOut_EP6002P2/D[14] <-> COM RxPDO-Map Outputs Channel 2/Data Out 14
//     PlcTask Outputs/GVL_IO.iq_stM3SelectorB.stComOut_EP6002P2/D[15] <-> COM RxPDO-Map Outputs Channel 2/Data Out 15
//     PlcTask Outputs/GVL_IO.iq_stM3SelectorB.stComOut_EP6002P2/D[16] <-> COM RxPDO-Map Outputs Channel 2/Data Out 16
//     PlcTask Outputs/GVL_IO.iq_stM3SelectorB.stComOut_EP6002P2/D[17] <-> COM RxPDO-Map Outputs Channel 2/Data Out 17
//     PlcTask Outputs/GVL_IO.iq_stM3SelectorB.stComOut_EP6002P2/D[18] <-> COM RxPDO-Map Outputs Channel 2/Data Out 18
//     PlcTask Outputs/GVL_IO.iq_stM3SelectorB.stComOut_EP6002P2/D[19] <-> COM RxPDO-Map Outputs Channel 2/Data Out 19
//     PlcTask Outputs/GVL_IO.iq_stM3SelectorB.stComOut_EP6002P2/D[1] <-> COM RxPDO-Map Outputs Channel 2/Data Out 1
//     PlcTask Outputs/GVL_IO.iq_stM3SelectorB.stComOut_EP6002P2/D[20] <-> COM RxPDO-Map Outputs Channel 2/Data Out 20
//     PlcTask Outputs/GVL_IO.iq_stM3SelectorB.stComOut_EP6002P2/D[21] <-> COM RxPDO-Map Outputs Channel 2/Data Out 21
//     PlcTask Outputs/GVL_IO.iq_stM3SelectorB.stComOut_EP6002P2/D[2] <-> COM RxPDO-Map Outputs Channel 2/Data Out 2
//     PlcTask Outputs/GVL_IO.iq_stM3SelectorB.stComOut_EP6002P2/D[3] <-> COM RxPDO-Map Outputs Channel 2/Data Out 3
//     PlcTask Outputs/GVL_IO.iq_stM3SelectorB.stComOut_EP6002P2/D[4] <-> COM RxPDO-Map Outputs Channel 2/Data Out 4
//     PlcTask Outputs/GVL_IO.iq_stM3SelectorB.stComOut_EP6002P2/D[5] <-> COM RxPDO-Map Outputs Channel 2/Data Out 5
//     PlcTask Outputs/GVL_IO.iq_stM3SelectorB.stComOut_EP6002P2/D[6] <-> COM RxPDO-Map Outputs Channel 2/Data Out 6
//     PlcTask Outputs/GVL_IO.iq_stM3SelectorB.stComOut_EP6002P2/D[7] <-> COM RxPDO-Map Outputs Channel 2/Data Out 7
//     PlcTask Outputs/GVL_IO.iq_stM3SelectorB.stComOut_EP6002P2/D[8] <-> COM RxPDO-Map Outputs Channel 2/Data Out 8
//     PlcTask Outputs/GVL_IO.iq_stM3SelectorB.stComOut_EP6002P2/D[9] <-> COM RxPDO-Map Outputs Channel 2/Data Out 9
//   SDSPLC Instance <-> MAIN (EtherCAT)/PCM A (EP3174-0002)
//     PlcTask Inputs/GVL_IO.iq_stPressCtrlA.i_EP3174_Ch{1..4} <-> AI Standard Channel {1..4}/Value  (4 links)
//   SDSPLC Instance <-> MAIN (EtherCAT)/PCM A (EP4374-0002)
//     PlcTask Inputs/GVL_IO.iq_stPressCtrlA.i_EP4374_Ch1 <-> AI Inputs Channel 1/Value
//     PlcTask Inputs/GVL_IO.iq_stPressCtrlA.i_EP4374_Ch2 <-> AI Inputs Channel 2/Value
//     PlcTask Outputs/GVL_IO.iq_stPressCtrlA.q_EP4374_Ch3 <-> AO Outputs Channel 3/Analog output
//     PlcTask Outputs/GVL_IO.iq_stPressCtrlA.q_EP4374_Ch4 <-> AO Outputs Channel 4/Analog output
//   SDSPLC Instance <-> MAIN (EtherCAT)/PCM A (EP6002-0002)
//     PlcTask Inputs/GVL_IO.iq_stPressCtrlA.stComIn_EP6002P1/D[0] <-> COM TxPDO-Map Inputs Channel 1/Data In 0
//     PlcTask Inputs/GVL_IO.iq_stPressCtrlA.stComIn_EP6002P1/D[10] <-> COM TxPDO-Map Inputs Channel 1/Data In 10
//     PlcTask Inputs/GVL_IO.iq_stPressCtrlA.stComIn_EP6002P1/D[11] <-> COM TxPDO-Map Inputs Channel 1/Data In 11
//     PlcTask Inputs/GVL_IO.iq_stPressCtrlA.stComIn_EP6002P1/D[12] <-> COM TxPDO-Map Inputs Channel 1/Data In 12
//     PlcTask Inputs/GVL_IO.iq_stPressCtrlA.stComIn_EP6002P1/D[13] <-> COM TxPDO-Map Inputs Channel 1/Data In 13
//     PlcTask Inputs/GVL_IO.iq_stPressCtrlA.stComIn_EP6002P1/D[14] <-> COM TxPDO-Map Inputs Channel 1/Data In 14
//     PlcTask Inputs/GVL_IO.iq_stPressCtrlA.stComIn_EP6002P1/D[15] <-> COM TxPDO-Map Inputs Channel 1/Data In 15
//     PlcTask Inputs/GVL_IO.iq_stPressCtrlA.stComIn_EP6002P1/D[16] <-> COM TxPDO-Map Inputs Channel 1/Data In 16
//     PlcTask Inputs/GVL_IO.iq_stPressCtrlA.stComIn_EP6002P1/D[17] <-> COM TxPDO-Map Inputs Channel 1/Data In 17
//     PlcTask Inputs/GVL_IO.iq_stPressCtrlA.stComIn_EP6002P1/D[18] <-> COM TxPDO-Map Inputs Channel 1/Data In 18
//     PlcTask Inputs/GVL_IO.iq_stPressCtrlA.stComIn_EP6002P1/D[19] <-> COM TxPDO-Map Inputs Channel 1/Data In 19
//     PlcTask Inputs/GVL_IO.iq_stPressCtrlA.stComIn_EP6002P1/D[1] <-> COM TxPDO-Map Inputs Channel 1/Data In 1
//     PlcTask Inputs/GVL_IO.iq_stPressCtrlA.stComIn_EP6002P1/D[20] <-> COM TxPDO-Map Inputs Channel 1/Data In 20
//     PlcTask Inputs/GVL_IO.iq_stPressCtrlA.stComIn_EP6002P1/D[21] <-> COM TxPDO-Map Inputs Channel 1/Data In 21
//     PlcTask Inputs/GVL_IO.iq_stPressCtrlA.stComIn_EP6002P1/D[2] <-> COM TxPDO-Map Inputs Channel 1/Data In 2
//     PlcTask Inputs/GVL_IO.iq_stPressCtrlA.stComIn_EP6002P1/D[3] <-> COM TxPDO-Map Inputs Channel 1/Data In 3
//     PlcTask Inputs/GVL_IO.iq_stPressCtrlA.stComIn_EP6002P1/D[4] <-> COM TxPDO-Map Inputs Channel 1/Data In 4
//     PlcTask Inputs/GVL_IO.iq_stPressCtrlA.stComIn_EP6002P1/D[5] <-> COM TxPDO-Map Inputs Channel 1/Data In 5
//     PlcTask Inputs/GVL_IO.iq_stPressCtrlA.stComIn_EP6002P1/D[6] <-> COM TxPDO-Map Inputs Channel 1/Data In 6
//     PlcTask Inputs/GVL_IO.iq_stPressCtrlA.stComIn_EP6002P1/D[7] <-> COM TxPDO-Map Inputs Channel 1/Data In 7
//     PlcTask Inputs/GVL_IO.iq_stPressCtrlA.stComIn_EP6002P1/D[8] <-> COM TxPDO-Map Inputs Channel 1/Data In 8
//     PlcTask Inputs/GVL_IO.iq_stPressCtrlA.stComIn_EP6002P1/D[9] <-> COM TxPDO-Map Inputs Channel 1/Data In 9
//     PlcTask Inputs/GVL_IO.iq_stPressCtrlA.stComIn_EP6002P2/D[0] <-> COM TxPDO-Map Inputs Channel 2/Data In 0
//     PlcTask Inputs/GVL_IO.iq_stPressCtrlA.stComIn_EP6002P2/D[10] <-> COM TxPDO-Map Inputs Channel 2/Data In 10
//     PlcTask Inputs/GVL_IO.iq_stPressCtrlA.stComIn_EP6002P2/D[11] <-> COM TxPDO-Map Inputs Channel 2/Data In 11
//     PlcTask Inputs/GVL_IO.iq_stPressCtrlA.stComIn_EP6002P2/D[12] <-> COM TxPDO-Map Inputs Channel 2/Data In 12
//     PlcTask Inputs/GVL_IO.iq_stPressCtrlA.stComIn_EP6002P2/D[13] <-> COM TxPDO-Map Inputs Channel 2/Data In 13
//     PlcTask Inputs/GVL_IO.iq_stPressCtrlA.stComIn_EP6002P2/D[14] <-> COM TxPDO-Map Inputs Channel 2/Data In 14
//     PlcTask Inputs/GVL_IO.iq_stPressCtrlA.stComIn_EP6002P2/D[15] <-> COM TxPDO-Map Inputs Channel 2/Data In 15
//     PlcTask Inputs/GVL_IO.iq_stPressCtrlA.stComIn_EP6002P2/D[16] <-> COM TxPDO-Map Inputs Channel 2/Data In 16
//     PlcTask Inputs/GVL_IO.iq_stPressCtrlA.stComIn_EP6002P2/D[17] <-> COM TxPDO-Map Inputs Channel 2/Data In 17
//     PlcTask Inputs/GVL_IO.iq_stPressCtrlA.stComIn_EP6002P2/D[18] <-> COM TxPDO-Map Inputs Channel 2/Data In 18
//     PlcTask Inputs/GVL_IO.iq_stPressCtrlA.stComIn_EP6002P2/D[19] <-> COM TxPDO-Map Inputs Channel 2/Data In 19
//     PlcTask Inputs/GVL_IO.iq_stPressCtrlA.stComIn_EP6002P2/D[1] <-> COM TxPDO-Map Inputs Channel 2/Data In 1
//     PlcTask Inputs/GVL_IO.iq_stPressCtrlA.stComIn_EP6002P2/D[20] <-> COM TxPDO-Map Inputs Channel 2/Data In 20
//     PlcTask Inputs/GVL_IO.iq_stPressCtrlA.stComIn_EP6002P2/D[21] <-> COM TxPDO-Map Inputs Channel 2/Data In 21
//     PlcTask Inputs/GVL_IO.iq_stPressCtrlA.stComIn_EP6002P2/D[2] <-> COM TxPDO-Map Inputs Channel 2/Data In 2
//     PlcTask Inputs/GVL_IO.iq_stPressCtrlA.stComIn_EP6002P2/D[3] <-> COM TxPDO-Map Inputs Channel 2/Data In 3
//     PlcTask Inputs/GVL_IO.iq_stPressCtrlA.stComIn_EP6002P2/D[4] <-> COM TxPDO-Map Inputs Channel 2/Data In 4
//     PlcTask Inputs/GVL_IO.iq_stPressCtrlA.stComIn_EP6002P2/D[5] <-> COM TxPDO-Map Inputs Channel 2/Data In 5
//     PlcTask Inputs/GVL_IO.iq_stPressCtrlA.stComIn_EP6002P2/D[6] <-> COM TxPDO-Map Inputs Channel 2/Data In 6
//     PlcTask Inputs/GVL_IO.iq_stPressCtrlA.stComIn_EP6002P2/D[7] <-> COM TxPDO-Map Inputs Channel 2/Data In 7
//     PlcTask Inputs/GVL_IO.iq_stPressCtrlA.stComIn_EP6002P2/D[8] <-> COM TxPDO-Map Inputs Channel 2/Data In 8
//     PlcTask Inputs/GVL_IO.iq_stPressCtrlA.stComIn_EP6002P2/D[9] <-> COM TxPDO-Map Inputs Channel 2/Data In 9
//     PlcTask Inputs/GVL_IO.iq_stPressCtrlA.stComIn_EP6002P1/Status <-> COM TxPDO-Map Inputs Channel 1/Status
//     PlcTask Inputs/GVL_IO.iq_stPressCtrlA.stComIn_EP6002P2/Status <-> COM TxPDO-Map Inputs Channel 2/Status
//     PlcTask Outputs/GVL_IO.iq_stPressCtrlA.stComOut_EP6002P1/Ctrl <-> COM RxPDO-Map Outputs Channel 1/Ctrl
//     PlcTask Outputs/GVL_IO.iq_stPressCtrlA.stComOut_EP6002P2/Ctrl <-> COM RxPDO-Map Outputs Channel 2/Ctrl
//     PlcTask Outputs/GVL_IO.iq_stPressCtrlA.stComOut_EP6002P1/D[0] <-> COM RxPDO-Map Outputs Channel 1/Data Out 0
//     PlcTask Outputs/GVL_IO.iq_stPressCtrlA.stComOut_EP6002P1/D[10] <-> COM RxPDO-Map Outputs Channel 1/Data Out 10
//     PlcTask Outputs/GVL_IO.iq_stPressCtrlA.stComOut_EP6002P1/D[11] <-> COM RxPDO-Map Outputs Channel 1/Data Out 11
//     PlcTask Outputs/GVL_IO.iq_stPressCtrlA.stComOut_EP6002P1/D[12] <-> COM RxPDO-Map Outputs Channel 1/Data Out 12
//     PlcTask Outputs/GVL_IO.iq_stPressCtrlA.stComOut_EP6002P1/D[13] <-> COM RxPDO-Map Outputs Channel 1/Data Out 13
//     PlcTask Outputs/GVL_IO.iq_stPressCtrlA.stComOut_EP6002P1/D[14] <-> COM RxPDO-Map Outputs Channel 1/Data Out 14
//     PlcTask Outputs/GVL_IO.iq_stPressCtrlA.stComOut_EP6002P1/D[15] <-> COM RxPDO-Map Outputs Channel 1/Data Out 15
//     PlcTask Outputs/GVL_IO.iq_stPressCtrlA.stComOut_EP6002P1/D[16] <-> COM RxPDO-Map Outputs Channel 1/Data Out 16
//     PlcTask Outputs/GVL_IO.iq_stPressCtrlA.stComOut_EP6002P1/D[17] <-> COM RxPDO-Map Outputs Channel 1/Data Out 17
//     PlcTask Outputs/GVL_IO.iq_stPressCtrlA.stComOut_EP6002P1/D[18] <-> COM RxPDO-Map Outputs Channel 1/Data Out 18
//     PlcTask Outputs/GVL_IO.iq_stPressCtrlA.stComOut_EP6002P1/D[19] <-> COM RxPDO-Map Outputs Channel 1/Data Out 19
//     PlcTask Outputs/GVL_IO.iq_stPressCtrlA.stComOut_EP6002P1/D[1] <-> COM RxPDO-Map Outputs Channel 1/Data Out 1
//     PlcTask Outputs/GVL_IO.iq_stPressCtrlA.stComOut_EP6002P1/D[20] <-> COM RxPDO-Map Outputs Channel 1/Data Out 20
//     PlcTask Outputs/GVL_IO.iq_stPressCtrlA.stComOut_EP6002P1/D[21] <-> COM RxPDO-Map Outputs Channel 1/Data Out 21
//     PlcTask Outputs/GVL_IO.iq_stPressCtrlA.stComOut_EP6002P1/D[2] <-> COM RxPDO-Map Outputs Channel 1/Data Out 2
//     PlcTask Outputs/GVL_IO.iq_stPressCtrlA.stComOut_EP6002P1/D[3] <-> COM RxPDO-Map Outputs Channel 1/Data Out 3
//     PlcTask Outputs/GVL_IO.iq_stPressCtrlA.stComOut_EP6002P1/D[4] <-> COM RxPDO-Map Outputs Channel 1/Data Out 4
//     PlcTask Outputs/GVL_IO.iq_stPressCtrlA.stComOut_EP6002P1/D[5] <-> COM RxPDO-Map Outputs Channel 1/Data Out 5
//     PlcTask Outputs/GVL_IO.iq_stPressCtrlA.stComOut_EP6002P1/D[6] <-> COM RxPDO-Map Outputs Channel 1/Data Out 6
//     PlcTask Outputs/GVL_IO.iq_stPressCtrlA.stComOut_EP6002P1/D[7] <-> COM RxPDO-Map Outputs Channel 1/Data Out 7
//     PlcTask Outputs/GVL_IO.iq_stPressCtrlA.stComOut_EP6002P1/D[8] <-> COM RxPDO-Map Outputs Channel 1/Data Out 8
//     PlcTask Outputs/GVL_IO.iq_stPressCtrlA.stComOut_EP6002P1/D[9] <-> COM RxPDO-Map Outputs Channel 1/Data Out 9
//     PlcTask Outputs/GVL_IO.iq_stPressCtrlA.stComOut_EP6002P2/D[0] <-> COM RxPDO-Map Outputs Channel 2/Data Out 0
//     PlcTask Outputs/GVL_IO.iq_stPressCtrlA.stComOut_EP6002P2/D[10] <-> COM RxPDO-Map Outputs Channel 2/Data Out 10
//     PlcTask Outputs/GVL_IO.iq_stPressCtrlA.stComOut_EP6002P2/D[11] <-> COM RxPDO-Map Outputs Channel 2/Data Out 11
//     PlcTask Outputs/GVL_IO.iq_stPressCtrlA.stComOut_EP6002P2/D[12] <-> COM RxPDO-Map Outputs Channel 2/Data Out 12
//     PlcTask Outputs/GVL_IO.iq_stPressCtrlA.stComOut_EP6002P2/D[13] <-> COM RxPDO-Map Outputs Channel 2/Data Out 13
//     PlcTask Outputs/GVL_IO.iq_stPressCtrlA.stComOut_EP6002P2/D[14] <-> COM RxPDO-Map Outputs Channel 2/Data Out 14
//     PlcTask Outputs/GVL_IO.iq_stPressCtrlA.stComOut_EP6002P2/D[15] <-> COM RxPDO-Map Outputs Channel 2/Data Out 15
//     PlcTask Outputs/GVL_IO.iq_stPressCtrlA.stComOut_EP6002P2/D[16] <-> COM RxPDO-Map Outputs Channel 2/Data Out 16
//     PlcTask Outputs/GVL_IO.iq_stPressCtrlA.stComOut_EP6002P2/D[17] <-> COM RxPDO-Map Outputs Channel 2/Data Out 17
//     PlcTask Outputs/GVL_IO.iq_stPressCtrlA.stComOut_EP6002P2/D[18] <-> COM RxPDO-Map Outputs Channel 2/Data Out 18
//     PlcTask Outputs/GVL_IO.iq_stPressCtrlA.stComOut_EP6002P2/D[19] <-> COM RxPDO-Map Outputs Channel 2/Data Out 19
//     PlcTask Outputs/GVL_IO.iq_stPressCtrlA.stComOut_EP6002P2/D[1] <-> COM RxPDO-Map Outputs Channel 2/Data Out 1
//     PlcTask Outputs/GVL_IO.iq_stPressCtrlA.stComOut_EP6002P2/D[20] <-> COM RxPDO-Map Outputs Channel 2/Data Out 20
//     PlcTask Outputs/GVL_IO.iq_stPressCtrlA.stComOut_EP6002P2/D[21] <-> COM RxPDO-Map Outputs Channel 2/Data Out 21
//     PlcTask Outputs/GVL_IO.iq_stPressCtrlA.stComOut_EP6002P2/D[2] <-> COM RxPDO-Map Outputs Channel 2/Data Out 2
//     PlcTask Outputs/GVL_IO.iq_stPressCtrlA.stComOut_EP6002P2/D[3] <-> COM RxPDO-Map Outputs Channel 2/Data Out 3
//     PlcTask Outputs/GVL_IO.iq_stPressCtrlA.stComOut_EP6002P2/D[4] <-> COM RxPDO-Map Outputs Channel 2/Data Out 4
//     PlcTask Outputs/GVL_IO.iq_stPressCtrlA.stComOut_EP6002P2/D[5] <-> COM RxPDO-Map Outputs Channel 2/Data Out 5
//     PlcTask Outputs/GVL_IO.iq_stPressCtrlA.stComOut_EP6002P2/D[6] <-> COM RxPDO-Map Outputs Channel 2/Data Out 6
//     PlcTask Outputs/GVL_IO.iq_stPressCtrlA.stComOut_EP6002P2/D[7] <-> COM RxPDO-Map Outputs Channel 2/Data Out 7
//     PlcTask Outputs/GVL_IO.iq_stPressCtrlA.stComOut_EP6002P2/D[8] <-> COM RxPDO-Map Outputs Channel 2/Data Out 8
//     PlcTask Outputs/GVL_IO.iq_stPressCtrlA.stComOut_EP6002P2/D[9] <-> COM RxPDO-Map Outputs Channel 2/Data Out 9
//   SDSPLC Instance <-> MAIN (EtherCAT)/PCM B (EP3174-0002)
//     PlcTask Inputs/GVL_IO.iq_stPressCtrlB.i_EP3174_Ch{1..4} <-> AI Standard Channel {1..4}/Value  (4 links)
//   SDSPLC Instance <-> MAIN (EtherCAT)/PCM B (EP4374-0002)
//     PlcTask Inputs/GVL_IO.iq_stPressCtrlB.i_EP4374_Ch1 <-> AI Inputs Channel 1/Value
//     PlcTask Inputs/GVL_IO.iq_stPressCtrlB.i_EP4374_Ch2 <-> AI Inputs Channel 2/Value
//     PlcTask Outputs/GVL_IO.iq_stPressCtrlB.q_EP4374_Ch3 <-> AO Outputs Channel 3/Analog output
//     PlcTask Outputs/GVL_IO.iq_stPressCtrlB.q_EP4374_Ch4 <-> AO Outputs Channel 4/Analog output
//   SDSPLC Instance <-> MAIN (EtherCAT)/PCM B (EP6002-0002)
//     PlcTask Inputs/GVL_IO.iq_stPressCtrlB.stComIn_EP6002P1/D[0] <-> COM TxPDO-Map Inputs Channel 1/Data In 0
//     PlcTask Inputs/GVL_IO.iq_stPressCtrlB.stComIn_EP6002P1/D[10] <-> COM TxPDO-Map Inputs Channel 1/Data In 10
//     PlcTask Inputs/GVL_IO.iq_stPressCtrlB.stComIn_EP6002P1/D[11] <-> COM TxPDO-Map Inputs Channel 1/Data In 11
//     PlcTask Inputs/GVL_IO.iq_stPressCtrlB.stComIn_EP6002P1/D[12] <-> COM TxPDO-Map Inputs Channel 1/Data In 12
//     PlcTask Inputs/GVL_IO.iq_stPressCtrlB.stComIn_EP6002P1/D[13] <-> COM TxPDO-Map Inputs Channel 1/Data In 13
//     PlcTask Inputs/GVL_IO.iq_stPressCtrlB.stComIn_EP6002P1/D[14] <-> COM TxPDO-Map Inputs Channel 1/Data In 14
//     PlcTask Inputs/GVL_IO.iq_stPressCtrlB.stComIn_EP6002P1/D[15] <-> COM TxPDO-Map Inputs Channel 1/Data In 15
//     PlcTask Inputs/GVL_IO.iq_stPressCtrlB.stComIn_EP6002P1/D[16] <-> COM TxPDO-Map Inputs Channel 1/Data In 16
//     PlcTask Inputs/GVL_IO.iq_stPressCtrlB.stComIn_EP6002P1/D[17] <-> COM TxPDO-Map Inputs Channel 1/Data In 17
//     PlcTask Inputs/GVL_IO.iq_stPressCtrlB.stComIn_EP6002P1/D[18] <-> COM TxPDO-Map Inputs Channel 1/Data In 18
//     PlcTask Inputs/GVL_IO.iq_stPressCtrlB.stComIn_EP6002P1/D[19] <-> COM TxPDO-Map Inputs Channel 1/Data In 19
//     PlcTask Inputs/GVL_IO.iq_stPressCtrlB.stComIn_EP6002P1/D[1] <-> COM TxPDO-Map Inputs Channel 1/Data In 1
//     PlcTask Inputs/GVL_IO.iq_stPressCtrlB.stComIn_EP6002P1/D[20] <-> COM TxPDO-Map Inputs Channel 1/Data In 20
//     PlcTask Inputs/GVL_IO.iq_stPressCtrlB.stComIn_EP6002P1/D[21] <-> COM TxPDO-Map Inputs Channel 1/Data In 21
//     PlcTask Inputs/GVL_IO.iq_stPressCtrlB.stComIn_EP6002P1/D[2] <-> COM TxPDO-Map Inputs Channel 1/Data In 2
//     PlcTask Inputs/GVL_IO.iq_stPressCtrlB.stComIn_EP6002P1/D[3] <-> COM TxPDO-Map Inputs Channel 1/Data In 3
//     PlcTask Inputs/GVL_IO.iq_stPressCtrlB.stComIn_EP6002P1/D[4] <-> COM TxPDO-Map Inputs Channel 1/Data In 4
//     PlcTask Inputs/GVL_IO.iq_stPressCtrlB.stComIn_EP6002P1/D[5] <-> COM TxPDO-Map Inputs Channel 1/Data In 5
//     PlcTask Inputs/GVL_IO.iq_stPressCtrlB.stComIn_EP6002P1/D[6] <-> COM TxPDO-Map Inputs Channel 1/Data In 6
//     PlcTask Inputs/GVL_IO.iq_stPressCtrlB.stComIn_EP6002P1/D[7] <-> COM TxPDO-Map Inputs Channel 1/Data In 7
//     PlcTask Inputs/GVL_IO.iq_stPressCtrlB.stComIn_EP6002P1/D[8] <-> COM TxPDO-Map Inputs Channel 1/Data In 8
//     PlcTask Inputs/GVL_IO.iq_stPressCtrlB.stComIn_EP6002P1/D[9] <-> COM TxPDO-Map Inputs Channel 1/Data In 9
//     PlcTask Inputs/GVL_IO.iq_stPressCtrlB.stComIn_EP6002P2/D[0] <-> COM TxPDO-Map Inputs Channel 2/Data In 0
//     PlcTask Inputs/GVL_IO.iq_stPressCtrlB.stComIn_EP6002P2/D[10] <-> COM TxPDO-Map Inputs Channel 2/Data In 10
//     PlcTask Inputs/GVL_IO.iq_stPressCtrlB.stComIn_EP6002P2/D[11] <-> COM TxPDO-Map Inputs Channel 2/Data In 11
//     PlcTask Inputs/GVL_IO.iq_stPressCtrlB.stComIn_EP6002P2/D[12] <-> COM TxPDO-Map Inputs Channel 2/Data In 12
//     PlcTask Inputs/GVL_IO.iq_stPressCtrlB.stComIn_EP6002P2/D[13] <-> COM TxPDO-Map Inputs Channel 2/Data In 13
//     PlcTask Inputs/GVL_IO.iq_stPressCtrlB.stComIn_EP6002P2/D[14] <-> COM TxPDO-Map Inputs Channel 2/Data In 14
//     PlcTask Inputs/GVL_IO.iq_stPressCtrlB.stComIn_EP6002P2/D[15] <-> COM TxPDO-Map Inputs Channel 2/Data In 15
//     PlcTask Inputs/GVL_IO.iq_stPressCtrlB.stComIn_EP6002P2/D[16] <-> COM TxPDO-Map Inputs Channel 2/Data In 16
//     PlcTask Inputs/GVL_IO.iq_stPressCtrlB.stComIn_EP6002P2/D[17] <-> COM TxPDO-Map Inputs Channel 2/Data In 17
//     PlcTask Inputs/GVL_IO.iq_stPressCtrlB.stComIn_EP6002P2/D[18] <-> COM TxPDO-Map Inputs Channel 2/Data In 18
//     PlcTask Inputs/GVL_IO.iq_stPressCtrlB.stComIn_EP6002P2/D[19] <-> COM TxPDO-Map Inputs Channel 2/Data In 19
//     PlcTask Inputs/GVL_IO.iq_stPressCtrlB.stComIn_EP6002P2/D[1] <-> COM TxPDO-Map Inputs Channel 2/Data In 1
//     PlcTask Inputs/GVL_IO.iq_stPressCtrlB.stComIn_EP6002P2/D[20] <-> COM TxPDO-Map Inputs Channel 2/Data In 20
//     PlcTask Inputs/GVL_IO.iq_stPressCtrlB.stComIn_EP6002P2/D[21] <-> COM TxPDO-Map Inputs Channel 2/Data In 21
//     PlcTask Inputs/GVL_IO.iq_stPressCtrlB.stComIn_EP6002P2/D[2] <-> COM TxPDO-Map Inputs Channel 2/Data In 2
//     PlcTask Inputs/GVL_IO.iq_stPressCtrlB.stComIn_EP6002P2/D[3] <-> COM TxPDO-Map Inputs Channel 2/Data In 3
//     PlcTask Inputs/GVL_IO.iq_stPressCtrlB.stComIn_EP6002P2/D[4] <-> COM TxPDO-Map Inputs Channel 2/Data In 4
//     PlcTask Inputs/GVL_IO.iq_stPressCtrlB.stComIn_EP6002P2/D[5] <-> COM TxPDO-Map Inputs Channel 2/Data In 5
//     PlcTask Inputs/GVL_IO.iq_stPressCtrlB.stComIn_EP6002P2/D[6] <-> COM TxPDO-Map Inputs Channel 2/Data In 6
//     PlcTask Inputs/GVL_IO.iq_stPressCtrlB.stComIn_EP6002P2/D[7] <-> COM TxPDO-Map Inputs Channel 2/Data In 7
//     PlcTask Inputs/GVL_IO.iq_stPressCtrlB.stComIn_EP6002P2/D[8] <-> COM TxPDO-Map Inputs Channel 2/Data In 8
//     PlcTask Inputs/GVL_IO.iq_stPressCtrlB.stComIn_EP6002P2/D[9] <-> COM TxPDO-Map Inputs Channel 2/Data In 9
//     PlcTask Inputs/GVL_IO.iq_stPressCtrlB.stComIn_EP6002P1/Status <-> COM TxPDO-Map Inputs Channel 1/Status
//     PlcTask Inputs/GVL_IO.iq_stPressCtrlB.stComIn_EP6002P2/Status <-> COM TxPDO-Map Inputs Channel 2/Status
//     PlcTask Outputs/GVL_IO.iq_stPressCtrlB.stComOut_EP6002P1/Ctrl <-> COM RxPDO-Map Outputs Channel 1/Ctrl
//     PlcTask Outputs/GVL_IO.iq_stPressCtrlB.stComOut_EP6002P2/Ctrl <-> COM RxPDO-Map Outputs Channel 2/Ctrl
//     PlcTask Outputs/GVL_IO.iq_stPressCtrlB.stComOut_EP6002P1/D[0] <-> COM RxPDO-Map Outputs Channel 1/Data Out 0
//     PlcTask Outputs/GVL_IO.iq_stPressCtrlB.stComOut_EP6002P1/D[10] <-> COM RxPDO-Map Outputs Channel 1/Data Out 10
//     PlcTask Outputs/GVL_IO.iq_stPressCtrlB.stComOut_EP6002P1/D[11] <-> COM RxPDO-Map Outputs Channel 1/Data Out 11
//     PlcTask Outputs/GVL_IO.iq_stPressCtrlB.stComOut_EP6002P1/D[12] <-> COM RxPDO-Map Outputs Channel 1/Data Out 12
//     PlcTask Outputs/GVL_IO.iq_stPressCtrlB.stComOut_EP6002P1/D[13] <-> COM RxPDO-Map Outputs Channel 1/Data Out 13
//     PlcTask Outputs/GVL_IO.iq_stPressCtrlB.stComOut_EP6002P1/D[14] <-> COM RxPDO-Map Outputs Channel 1/Data Out 14
//     PlcTask Outputs/GVL_IO.iq_stPressCtrlB.stComOut_EP6002P1/D[15] <-> COM RxPDO-Map Outputs Channel 1/Data Out 15
//     PlcTask Outputs/GVL_IO.iq_stPressCtrlB.stComOut_EP6002P1/D[16] <-> COM RxPDO-Map Outputs Channel 1/Data Out 16
//     PlcTask Outputs/GVL_IO.iq_stPressCtrlB.stComOut_EP6002P1/D[17] <-> COM RxPDO-Map Outputs Channel 1/Data Out 17
//     PlcTask Outputs/GVL_IO.iq_stPressCtrlB.stComOut_EP6002P1/D[18] <-> COM RxPDO-Map Outputs Channel 1/Data Out 18
//     PlcTask Outputs/GVL_IO.iq_stPressCtrlB.stComOut_EP6002P1/D[19] <-> COM RxPDO-Map Outputs Channel 1/Data Out 19
//     PlcTask Outputs/GVL_IO.iq_stPressCtrlB.stComOut_EP6002P1/D[1] <-> COM RxPDO-Map Outputs Channel 1/Data Out 1
//     PlcTask Outputs/GVL_IO.iq_stPressCtrlB.stComOut_EP6002P1/D[20] <-> COM RxPDO-Map Outputs Channel 1/Data Out 20
//     PlcTask Outputs/GVL_IO.iq_stPressCtrlB.stComOut_EP6002P1/D[21] <-> COM RxPDO-Map Outputs Channel 1/Data Out 21
//     PlcTask Outputs/GVL_IO.iq_stPressCtrlB.stComOut_EP6002P1/D[2] <-> COM RxPDO-Map Outputs Channel 1/Data Out 2
//     PlcTask Outputs/GVL_IO.iq_stPressCtrlB.stComOut_EP6002P1/D[3] <-> COM RxPDO-Map Outputs Channel 1/Data Out 3
//     PlcTask Outputs/GVL_IO.iq_stPressCtrlB.stComOut_EP6002P1/D[4] <-> COM RxPDO-Map Outputs Channel 1/Data Out 4
//     PlcTask Outputs/GVL_IO.iq_stPressCtrlB.stComOut_EP6002P1/D[5] <-> COM RxPDO-Map Outputs Channel 1/Data Out 5
//     PlcTask Outputs/GVL_IO.iq_stPressCtrlB.stComOut_EP6002P1/D[6] <-> COM RxPDO-Map Outputs Channel 1/Data Out 6
//     PlcTask Outputs/GVL_IO.iq_stPressCtrlB.stComOut_EP6002P1/D[7] <-> COM RxPDO-Map Outputs Channel 1/Data Out 7
//     PlcTask Outputs/GVL_IO.iq_stPressCtrlB.stComOut_EP6002P1/D[8] <-> COM RxPDO-Map Outputs Channel 1/Data Out 8
//     PlcTask Outputs/GVL_IO.iq_stPressCtrlB.stComOut_EP6002P1/D[9] <-> COM RxPDO-Map Outputs Channel 1/Data Out 9
//     PlcTask Outputs/GVL_IO.iq_stPressCtrlB.stComOut_EP6002P2/D[0] <-> COM RxPDO-Map Outputs Channel 2/Data Out 0
//     PlcTask Outputs/GVL_IO.iq_stPressCtrlB.stComOut_EP6002P2/D[10] <-> COM RxPDO-Map Outputs Channel 2/Data Out 10
//     PlcTask Outputs/GVL_IO.iq_stPressCtrlB.stComOut_EP6002P2/D[11] <-> COM RxPDO-Map Outputs Channel 2/Data Out 11
//     PlcTask Outputs/GVL_IO.iq_stPressCtrlB.stComOut_EP6002P2/D[12] <-> COM RxPDO-Map Outputs Channel 2/Data Out 12
//     PlcTask Outputs/GVL_IO.iq_stPressCtrlB.stComOut_EP6002P2/D[13] <-> COM RxPDO-Map Outputs Channel 2/Data Out 13
//     PlcTask Outputs/GVL_IO.iq_stPressCtrlB.stComOut_EP6002P2/D[14] <-> COM RxPDO-Map Outputs Channel 2/Data Out 14
//     PlcTask Outputs/GVL_IO.iq_stPressCtrlB.stComOut_EP6002P2/D[15] <-> COM RxPDO-Map Outputs Channel 2/Data Out 15
//     PlcTask Outputs/GVL_IO.iq_stPressCtrlB.stComOut_EP6002P2/D[16] <-> COM RxPDO-Map Outputs Channel 2/Data Out 16
//     PlcTask Outputs/GVL_IO.iq_stPressCtrlB.stComOut_EP6002P2/D[17] <-> COM RxPDO-Map Outputs Channel 2/Data Out 17
//     PlcTask Outputs/GVL_IO.iq_stPressCtrlB.stComOut_EP6002P2/D[18] <-> COM RxPDO-Map Outputs Channel 2/Data Out 18
//     PlcTask Outputs/GVL_IO.iq_stPressCtrlB.stComOut_EP6002P2/D[19] <-> COM RxPDO-Map Outputs Channel 2/Data Out 19
//     PlcTask Outputs/GVL_IO.iq_stPressCtrlB.stComOut_EP6002P2/D[1] <-> COM RxPDO-Map Outputs Channel 2/Data Out 1
//     PlcTask Outputs/GVL_IO.iq_stPressCtrlB.stComOut_EP6002P2/D[20] <-> COM RxPDO-Map Outputs Channel 2/Data Out 20
//     PlcTask Outputs/GVL_IO.iq_stPressCtrlB.stComOut_EP6002P2/D[21] <-> COM RxPDO-Map Outputs Channel 2/Data Out 21
//     PlcTask Outputs/GVL_IO.iq_stPressCtrlB.stComOut_EP6002P2/D[2] <-> COM RxPDO-Map Outputs Channel 2/Data Out 2
//     PlcTask Outputs/GVL_IO.iq_stPressCtrlB.stComOut_EP6002P2/D[3] <-> COM RxPDO-Map Outputs Channel 2/Data Out 3
//     PlcTask Outputs/GVL_IO.iq_stPressCtrlB.stComOut_EP6002P2/D[4] <-> COM RxPDO-Map Outputs Channel 2/Data Out 4
//     PlcTask Outputs/GVL_IO.iq_stPressCtrlB.stComOut_EP6002P2/D[5] <-> COM RxPDO-Map Outputs Channel 2/Data Out 5
//     PlcTask Outputs/GVL_IO.iq_stPressCtrlB.stComOut_EP6002P2/D[6] <-> COM RxPDO-Map Outputs Channel 2/Data Out 6
//     PlcTask Outputs/GVL_IO.iq_stPressCtrlB.stComOut_EP6002P2/D[7] <-> COM RxPDO-Map Outputs Channel 2/Data Out 7
//     PlcTask Outputs/GVL_IO.iq_stPressCtrlB.stComOut_EP6002P2/D[8] <-> COM RxPDO-Map Outputs Channel 2/Data Out 8
//     PlcTask Outputs/GVL_IO.iq_stPressCtrlB.stComOut_EP6002P2/D[9] <-> COM RxPDO-Map Outputs Channel 2/Data Out 9
//   SDSPLC Instance <-> NC-Task 1 SAF/Axes/ALI_PropValve
//     PlcTask Inputs/GVL_Devices.stALI.stPropVlv.stAxis.NcToPlc <-> Outputs/ToPlc
//     PlcTask Outputs/GVL_Devices.stALI.stPropVlv.stAxis.PlcToNc <-> Inputs/FromPlc
//   SDSPLC Instance <-> NC-Task 1 SAF/Axes/ALI_X
//     PlcTask Inputs/GVL_Devices.stALI.axisX.stAxis.NcToPlc <-> Outputs/ToPlc
//     PlcTask Outputs/GVL_Devices.stALI.axisX.stAxis.PlcToNc <-> Inputs/FromPlc
//   SDSPLC Instance <-> NC-Task 1 SAF/Axes/ALI_Y
//     PlcTask Inputs/GVL_Devices.stALI.axisY.stAxis.NcToPlc <-> Outputs/ToPlc
//     PlcTask Outputs/GVL_Devices.stALI.axisY.stAxis.PlcToNc <-> Inputs/FromPlc
//   SDSPLC Instance <-> NC-Task 1 SAF/Axes/ALI_Z
//     PlcTask Inputs/GVL_Devices.stALI.axisZ.stAxis.NcToPlc <-> Outputs/ToPlc
//     PlcTask Outputs/GVL_Devices.stALI.axisZ.stAxis.PlcToNc <-> Inputs/FromPlc

// ---- POUs/VICI/FB_ViciDriver.TcPOU
FUNCTION_BLOCK FB_ViciDriver
FUNCTION_BLOCK FB_ViciDriver
VAR_INPUT
	i_xExecute				: BOOL;					(* rising edge execute *)
	i_tTimeOut				: TIME := t#10s;  		(* Maximum wait time for reply *)
	i_stControl				: ST_ViciControl;
END_VAR
VAR_OUTPUT
	q_xDone					: BOOL;
	q_xError				: BOOL;
	q_xWarning				: BOOL;					(* set in the event of an unexpected reply *)
	q_xTimeout				: BOOL;
	q_sResult				: STRING(255);
	q_sLastSentString		: ARRAY[1..40] OF STRING;				(* Last String Sent to Serial Device - for debugging *)
	q_sLastReceivedString	: ARRAY[1..40] OF STRING;				(* Last String Received from Serial Device - for debugging *)
	q_stStatus				: ST_ViciStatus;
END_VAR
VAR_IN_OUT
	iq_stSerialRXBuffer 	: ComBuffer;
	iq_stSerialTXBuffer 	: ComBuffer;
END_VAR
VAR
	rtExecute				: R_TRIG;
	iStep					: INT;
	sSendData				: STRING;
	fbViciTransaction		: FB_ViciTransaction;
	(*fbFormatString			: FB_FormatString;*)
	(*fbSplit					: FB_Split255;*)
	asReplyFields			: ARRAY[1..20] OF T_MaxString;
	wChecksum: WORD;
	rtStartIntegration: R_TRIG;
	rtEndReset: R_TRIG;

	sWorking: STRING;
	strResponseExpected: STRING;
END_VAR

(* This function block performs serial transactions with a Vici *)

(* rising edge trigger *)
rtExecute(CLK:= i_xExecute);
IF rtExecute.Q  THEN
	q_xDone	:= FALSE;
	q_xError := FALSE;
	q_xWarning := FALSE;
	q_xTimeout := FALSE;
	q_sResult:= '';
	FBViciTransaction( i_xExecute:= FALSE, iq_stSerialRXBuffer:= iq_stSerialRXBuffer, iq_stSerialTXBuffer:= iq_stSerialTXBuffer );  (* reset *)
	iStep := 10;
END_IF

CASE iStep OF
	0: (* idle *)
		;

	10: (* Get Position *)
		FBViciTransaction(
			i_xExecute:= TRUE,
			i_iAddress:=i_stControl.iAddress,
			i_sSendData:= 'CP', (*declared postion readback Vici command*)
			i_tTimeOut:= i_tTimeOut,
			iq_stSerialRXBuffer:= iq_stSerialRXBuffer,
			iq_stSerialTXBuffer:= iq_stSerialTXBuffer,
			i_CmdFlag :=FALSE);
		IF FBViciTransaction.q_xError THEN
			q_sResult := CONCAT('in Step 10 serial transaction failed with message: ', FBViciTransaction.q_sResult);
			q_stStatus.xPosValid := FALSE; (* used to signal an invalid readback or control exchange *)
			iStep := 9000;
		ELSIF FBViciTransaction.q_xDone THEN
			q_stStatus.sViciReply := FBViciTransaction.q_sResponseData;
			(* grab the left two characters, they should equal CP *)
			strResponseExpected := CONCAT(INT_TO_STRING( i_stControl.iAddress), 'CP');
			IF LEFT(q_stStatus.sViciReply, 3) <> strResponseExpected (*'1CP'*) THEN
				(*use q-s Result to specify error type*)
				q_sResult := CONCAT(CONCAT('in step 10 unexpected response recieved: ', LEFT(q_stStatus.sViciReply, 3)),CONCAT(' instead of: ', CONCAT(INT_TO_STRING( i_stControl.iAddress), 'CP')));
					q_xWarning := TRUE;
				(* If they don't equal CP, then error *)
				q_stStatus.xPosValid := FALSE; (* used to signal an invalid readback or control exchange *)
				iStep := 9000;
			(* else then grab the right two characters and convert to INT *)
			ELSE
			sWorking := RIGHT(q_stStatus.sViciReply, 2);
			q_stStatus.iCurrPos (* pass that INT to the q_stStatus.iCurrPos *) := STRING_TO_INT(sWorking);
			q_stStatus.xPosValid := TRUE;
			FBViciTransaction( i_xExecute:= FALSE, iq_stSerialRXBuffer:= iq_stSerialRXBuffer, iq_stSerialTXBuffer:= iq_stSerialTXBuffer, i_CmdFlag :=FALSE);  (* reset *)
			iStep := 5000;
			END_IF
		END_IF


	5000: (* Set position*)
		IF q_stStatus.iReqPos <> i_stControl.iReqPos THEN
			(*noah's code *)
			IF i_stControl.iReqPos > 12 OR i_stControl.iReqPos < 1 THEN
				q_sResult := CONCAT('in step 5000 port range exceeded: ',FBViciTransaction.q_sResponseData);
				i_stControl.iReqPos := LIMIT(1, i_stControl.iReqPos,12);
			ELSIF q_stStatus.iCurrPos > i_stControl.iReqPos THEN
				sSendData := CONCAT('CW', INT_TO_STRING(i_stControl.iReqPos));
			ELSE
				sSendData := CONCAT('CC', INT_TO_STRING(i_stControl.iReqPos));
			END_IF
			FBViciTransaction(
				i_xExecute:= TRUE,
				i_sSendData:= sSendData,
				i_tTimeOut:= i_tTimeOut,
				i_iAddress:=i_stControl.iAddress,
				iq_stSerialRXBuffer:= iq_stSerialRXBuffer,
				iq_stSerialTXBuffer:= iq_stSerialTXBuffer,
				i_CmdFlag:=TRUE);
			IF FBViciTransaction.q_xError THEN
				q_sResult := CONCAT('in Step 5000 serial transaction failed with message: ', FBViciTransaction.q_sResult);
				iStep := 9000;
			ELSIF FBViciTransaction.q_xDone THEN
				FBViciTransaction(
					 i_xExecute:= FALSE,
					iq_stSerialRXBuffer:= iq_stSerialRXBuffer,
					iq_stSerialTXBuffer:= iq_stSerialTXBuffer,
					i_CmdFlag:=FALSE );  (* reset *)
				q_stStatus.iReqPos := i_stControl.iReqPos;
				iStep := 8000;
			END_IF
		ELSE
			iStep := 8000;
		END_IF


	8000: (* done *)
		q_xDone := TRUE;
		IF q_sResult = '' THEN
			q_sResult := 'Success';
		END_IF
		IF  i_xExecute = FALSE THEN
			q_xDone:= FALSE;
			iStep := 0;
		END_IF

	9000:
		_A_ClearStatus();
		q_xTimeout := FBViciTransaction.q_xTimeout;
		q_xError := TRUE;
		

END_CASE

q_sLastSentString := FBViciTransaction.q_sLastSentString;
q_sLastReceivedString := FBViciTransaction.q_sLastReceivedString;

ACTION _A_ClearStatus:
q_stStatus.sViciReply := '';
END_ACTION

END_FUNCTION_BLOCK
